LIN {X 88.798,Y 87.967,Z 72.038,A 180.000,B 0.000,C 180.000} C_DIS
LIN {X 88.452,Y 88.283,Z 72.022,A 180.000,B 0.000,C 180.000} C_DIS
LIN {X 88.396,Y 88.335,Z 72.019,A 180.000,B 0.000,C 180.000} C_DIS
LIN {X 88.341,Y 88.389,Z 72.016,A 180.000,B 0.000,C 180.000} C_DIS
LIN {X 88.287,Y 88.444,Z 72.014,A 180.000,B 0.000,C 180.000} C_DIS
LIN {X 87.963,Y 88.776,Z 71.998,A 180.000,B 0.000,C 180.000} C_DIS
LIN {X 87.909,Y 88.831,Z 71.995,A 180.000,B 0.000,C 180.000} C_DIS
LIN {X 87.856,Y 88.887,Z 71.992,A 180.000,B 0.000,C 180.000} C_DIS
LIN {X 87.804,Y 88.944,Z 71.990,A 180.000,B 0.000,C 180.000} C_DIS
LIN {X 87.702,Y 89.060,Z 71.984,A 180.000,B 0.000,C 180.000} C_DIS
LIN {X 87.445,Y 89.355,Z 71.970,A 180.000,B 0.000,C 180.000} C_DIS
LIN {X 87.396,Y 89.412,Z 71.968,A 180.000,B 0.000,C 180.000} C_DIS
LIN {X 87.349,Y 89.471,Z 71.965,A 180.000,B 0.000,C 180.000} C_DIS
LIN {X 87.254,Y 89.593,Z 71.960,A 180.000,B 0.000,C 180.000} C_DIS
LIN {X 87.013,Y 89.903,Z 71.946,A 180.000,B 0.000,C 180.000} C_DIS
LIN {X 86.965,Y 89.965,Z 71.943,A 180.000,B 0.000,C 180.000} C_DIS
LIN {X 86.918,Y 90.027,Z 71.941,A 180.000,B 0.000,C 180.000} C_DIS
LIN {X 86.874,Y 90.090,Z 71.938,A 180.000,B 0.000,C 180.000} C_DIS
LIN {X 86.564,Y 90.537,Z 71.919,A 180.000,B 0.000,C 180.000} C_DIS
LIN {X 86.522,Y 90.601,Z 71.916,A 180.000,B 0.000,C 180.000} C_DIS
LIN {X 86.481,Y 90.665,Z 71.914,A 180.000,B 0.000,C 180.000} C_DIS
LIN {X 86.197,Y 91.129,Z 71.895,A 180.000,B 0.000,C 180.000} C_DIS
LIN {X 86.158,Y 91.194,Z 71.892,A 180.000,B 0.000,C 180.000} C_DIS
LIN {X 86.121,Y 91.260,Z 71.889,A 180.000,B 0.000,C 180.000} C_DIS
LIN {X 86.084,Y 91.327,Z 71.887,A 180.000,B 0.000,C 180.000} C_DIS
LIN {X 85.972,Y 91.535,Z 71.878,A 180.000,B 0.000,C 180.000} C_DIS
LIN {X 85.898,Y 91.673,Z 71.873,A 180.000,B 0.000,C 180.000} C_DIS
LIN {X 85.824,Y 91.810,Z 71.868,A 180.000,B 0.000,C 180.000} C_DIS
LIN {X 85.789,Y 91.879,Z 71.865,A 180.000,B 0.000,C 180.000} C_DIS
LIN {X 85.755,Y 91.949,Z 71.862,A 180.000,B 0.000,C 180.000} C_DIS
LIN {X 85.557,Y 92.373,Z 71.846,A 180.000,B 0.000,C 180.000} C_DIS
LIN {X 85.524,Y 92.444,Z 71.843,A 180.000,B 0.000,C 180.000} C_DIS
LIN {X 85.493,Y 92.514,Z 71.840,A 180.000,B 0.000,C 180.000} C_DIS
LIN {X 85.463,Y 92.585,Z 71.838,A 180.000,B 0.000,C 180.000} C_DIS
LIN {X 85.435,Y 92.656,Z 71.835,A 180.000,B 0.000,C 180.000} C_DIS
LIN {X 85.406,Y 92.727,Z 71.832,A 180.000,B 0.000,C 180.000} C_DIS
LIN {X 85.348,Y 92.873,Z 71.827,A 180.000,B 0.000,C 180.000} C_DIS
LIN {X 85.260,Y 93.091,Z 71.819,A 180.000,B 0.000,C 180.000} C_DIS
LIN {X 85.232,Y 93.163,Z 71.816,A 180.000,B 0.000,C 180.000} C_DIS
LIN {X 85.205,Y 93.235,Z 71.813,A 180.000,B 0.000,C 180.000} C_DIS
LIN {X 85.180,Y 93.308,Z 71.811,A 180.000,B 0.000,C 180.000} C_DIS
LIN {X 85.130,Y 93.456,Z 71.805,A 180.000,B 0.000,C 180.000} C_DIS
LIN {X 85.030,Y 93.751,Z 71.794,A 180.000,B 0.000,C 180.000} C_DIS
LIN {X 85.006,Y 93.825,Z 71.792,A 180.000,B 0.000,C 180.000} C_DIS
LIN {X 84.982,Y 93.898,Z 71.789,A 180.000,B 0.000,C 180.000} C_DIS
LIN {X 84.961,Y 93.974,Z 71.786,A 180.000,B 0.000,C 180.000} C_DIS
LIN {X 84.920,Y 94.125,Z 71.781,A 180.000,B 0.000,C 180.000} C_DIS
LIN {X 84.899,Y 94.200,Z 71.778,A 180.000,B 0.000,C 180.000} C_DIS
LIN {X 84.857,Y 94.352,Z 71.772,A 180.000,B 0.000,C 180.000} C_DIS
LIN {X 84.836,Y 94.428,Z 71.770,A 180.000,B 0.000,C 180.000} C_DIS
LIN {X 84.815,Y 94.504,Z 71.767,A 180.000,B 0.000,C 180.000} C_DIS
LIN {X 84.795,Y 94.578,Z 71.764,A 180.000,B 0.000,C 180.000} C_DIS
LIN {X 84.777,Y 94.653,Z 71.761,A 180.000,B 0.000,C 180.000} C_DIS
LIN {X 84.760,Y 94.728,Z 71.759,A 180.000,B 0.000,C 180.000} C_DIS
LIN {X 84.744,Y 94.804,Z 71.756,A 180.000,B 0.000,C 180.000} C_DIS
LIN {X 84.711,Y 94.958,Z 71.751,A 180.000,B 0.000,C 180.000} C_DIS
LIN {X 84.661,Y 95.187,Z 71.742,A 180.000,B 0.000,C 180.000} C_DIS
LIN {X 84.645,Y 95.263,Z 71.740,A 180.000,B 0.000,C 180.000} C_DIS
LIN {X 84.631,Y 95.339,Z 71.737,A 180.000,B 0.000,C 180.000} C_DIS
LIN {X 84.618,Y 95.415,Z 71.734,A 180.000,B 0.000,C 180.000} C_DIS
LIN {X 84.594,Y 95.571,Z 71.729,A 180.000,B 0.000,C 180.000} C_DIS
LIN {X 84.557,Y 95.803,Z 71.721,A 180.000,B 0.000,C 180.000} C_DIS
LIN {X 84.545,Y 95.880,Z 71.718,A 180.000,B 0.000,C 180.000} C_DIS
LIN {X 84.533,Y 95.956,Z 71.715,A 180.000,B 0.000,C 180.000} C_DIS
LIN {X 84.522,Y 96.033,Z 71.712,A 180.000,B 0.000,C 180.000} C_DIS
LIN {X 84.512,Y 96.111,Z 71.710,A 180.000,B 0.000,C 180.000} C_DIS
LIN {X 84.504,Y 96.189,Z 71.707,A 180.000,B 0.000,C 180.000} C_DIS
LIN {X 84.481,Y 96.424,Z 71.699,A 180.000,B 0.000,C 180.000} C_DIS
LIN {X 84.465,Y 96.580,Z 71.693,A 180.000,B 0.000,C 180.000} C_DIS
LIN {X 84.457,Y 96.659,Z 71.691,A 180.000,B 0.000,C 180.000} C_DIS
LIN {X 84.450,Y 96.736,Z 71.688,A 180.000,B 0.000,C 180.000} C_DIS
LIN {X 84.444,Y 96.813,Z 71.685,A 180.000,B 0.000,C 180.000} C_DIS
LIN {X 84.441,Y 96.891,Z 71.683,A 180.000,B 0.000,C 180.000} C_DIS
LIN {X 84.431,Y 97.125,Z 71.675,A 180.000,B 0.000,C 180.000} C_DIS
LIN {X 84.427,Y 97.204,Z 71.672,A 180.000,B 0.000,C 180.000} C_DIS
LIN {X 84.424,Y 97.283,Z 71.669,A 180.000,B 0.000,C 180.000} C_DIS
LIN {X 84.420,Y 97.361,Z 71.667,A 180.000,B 0.000,C 180.000} C_DIS
LIN {X 84.417,Y 97.439,Z 71.664,A 180.000,B 0.000,C 180.000} C_DIS
LIN {X 84.416,Y 97.517,Z 71.662,A 180.000,B 0.000,C 180.000} C_DIS
LIN {X 84.416,Y 97.595,Z 71.659,A 180.000,B 0.000,C 180.000} C_DIS
LIN {X 84.417,Y 97.674,Z 71.656,A 180.000,B 0.000,C 180.000} C_DIS
LIN {X 84.418,Y 97.752,Z 71.654,A 180.000,B 0.000,C 180.000} C_DIS
LIN {X 84.419,Y 97.830,Z 71.651,A 180.000,B 0.000,C 180.000} C_DIS
LIN {X 84.420,Y 97.909,Z 71.649,A 180.000,B 0.000,C 180.000} C_DIS
LIN {X 84.422,Y 98.065,Z 71.644,A 180.000,B 0.000,C 180.000} C_DIS
LIN {X 84.424,Y 98.222,Z 71.639,A 180.000,B 0.000,C 180.000} C_DIS
LIN {X 84.434,Y 98.378,Z 71.634,A 180.000,B 0.000,C 180.000} C_DIS
LIN {X 84.445,Y 98.534,Z 71.630,A 180.000,B 0.000,C 180.000} C_DIS
LIN {X 84.456,Y 98.691,Z 71.625,A 180.000,B 0.000,C 180.000} C_DIS
LIN {X 84.467,Y 98.849,Z 71.620,A 180.000,B 0.000,C 180.000} C_DIS
LIN {X 84.481,Y 99.004,Z 71.616,A 180.000,B 0.000,C 180.000} C_DIS
LIN {X 84.500,Y 99.159,Z 71.611,A 180.000,B 0.000,C 180.000} C_DIS
LIN {X 84.520,Y 99.315,Z 71.607,A 180.000,B 0.000,C 180.000} C_DIS
LIN {X 84.540,Y 99.471,Z 71.602,A 180.000,B 0.000,C 180.000} C_DIS
LIN {X 84.560,Y 99.626,Z 71.598,A 180.000,B 0.000,C 180.000} C_DIS
LIN {X 84.584,Y 99.781,Z 71.594,A 180.000,B 0.000,C 180.000} C_DIS
LIN {X 84.613,Y 99.935,Z 71.590,A 180.000,B 0.000,C 180.000} C_DIS
LIN {X 84.642,Y 100.090,Z 71.586,A 180.000,B 0.000,C 180.000} C_DIS
LIN {X 84.671,Y 100.245,Z 71.582,A 180.000,B 0.000,C 180.000} C_DIS
LIN {X 84.700,Y 100.399,Z 71.578,A 180.000,B 0.000,C 180.000} C_DIS
LIN {X 84.737,Y 100.552,Z 71.574,A 180.000,B 0.000,C 180.000} C_DIS
LIN {X 84.774,Y 100.704,Z 71.570,A 180.000,B 0.000,C 180.000} C_DIS
LIN {X 84.812,Y 100.857,Z 71.567,A 180.000,B 0.000,C 180.000} C_DIS
LIN {X 84.850,Y 101.009,Z 71.563,A 180.000,B 0.000,C 180.000} C_DIS
LIN {X 84.888,Y 101.161,Z 71.560,A 180.000,B 0.000,C 180.000} C_DIS
LIN {X 84.934,Y 101.312,Z 71.556,A 180.000,B 0.000,C 180.000} C_DIS
LIN {X 84.980,Y 101.462,Z 71.553,A 180.000,B 0.000,C 180.000} C_DIS
LIN {X 85.027,Y 101.613,Z 71.550,A 180.000,B 0.000,C 180.000} C_DIS
LIN {X 85.073,Y 101.763,Z 71.547,A 180.000,B 0.000,C 180.000} C_DIS
LIN {X 85.124,Y 101.911,Z 71.544,A 180.000,B 0.000,C 180.000} C_DIS
LIN {X 85.179,Y 102.059,Z 71.541,A 180.000,B 0.000,C 180.000} C_DIS
LIN {X 85.234,Y 102.206,Z 71.538,A 180.000,B 0.000,C 180.000} C_DIS
LIN {X 85.289,Y 102.354,Z 71.535,A 180.000,B 0.000,C 180.000} C_DIS
LIN {X 85.344,Y 102.501,Z 71.532,A 180.000,B 0.000,C 180.000} C_DIS
LIN {X 85.405,Y 102.646,Z 71.530,A 180.000,B 0.000,C 180.000} C_DIS
LIN {X 85.468,Y 102.790,Z 71.527,A 180.000,B 0.000,C 180.000} C_DIS
LIN {X 85.594,Y 103.079,Z 71.523,A 180.000,B 0.000,C 180.000} C_DIS
LIN {X 85.730,Y 103.362,Z 71.519,A 180.000,B 0.000,C 180.000} C_DIS
LIN {X 85.873,Y 103.643,Z 71.515,A 180.000,B 0.000,C 180.000} C_DIS
LIN {X 86.020,Y 103.921,Z 71.511,A 180.000,B 0.000,C 180.000} C_DIS
LIN {X 86.178,Y 104.193,Z 71.508,A 180.000,B 0.000,C 180.000} C_DIS
LIN {X 86.337,Y 104.465,Z 71.506,A 180.000,B 0.000,C 180.000} C_DIS
LIN {X 86.509,Y 104.729,Z 71.504,A 180.000,B 0.000,C 180.000} C_DIS
LIN {X 86.684,Y 104.991,Z 71.502,A 180.000,B 0.000,C 180.000} C_DIS
LIN {X 86.866,Y 105.248,Z 71.501,A 180.000,B 0.000,C 180.000} C_DIS
LIN {X 87.055,Y 105.500,Z 71.500,A 180.000,B 0.000,C 180.000} C_DIS
LIN {X 87.227,Y 105.724,Z 71.500,A 180.000,B 0.000,C 180.000} C_DIS
; Cutting Move Starts
LIN {X 87.243,Y 105.745,Z 71.500,A 180.000,B 0.000,C 180.000} C_DIS
LIN {X 87.319,Y 105.835,Z 71.500,A 180.000,B 0.000,C 180.000} C_DIS
LIN {X 87.621,Y 106.193,Z 71.500,A 180.000,B 0.000,C 180.000} C_DIS
LIN {X 87.779,Y 106.367,Z 71.500,A 180.000,B 0.000,C 180.000} C_DIS
LIN {X 88.137,Y 106.746,Z 71.500,A 180.000,B 0.000,C 180.000} C_DIS
LIN {X 88.300,Y 106.908,Z 71.500,A 180.000,B 0.000,C 180.000} C_DIS
LIN {X 88.673,Y 107.260,Z 71.500,A 180.000,B 0.000,C 180.000} C_DIS
LIN {X 88.678,Y 107.265,Z 71.500,A 180.000,B 0.000,C 180.000} C_DIS
LIN {X 88.852,Y 107.416,Z 71.500,A 180.000,B 0.000,C 180.000} C_DIS
LIN {X 89.209,Y 107.718,Z 71.500,A 180.000,B 0.000,C 180.000} C_DIS
LIN {X 89.311,Y 107.802,Z 71.500,A 180.000,B 0.000,C 180.000} C_DIS
LIN {X 89.388,Y 107.861,Z 71.500,A 180.000,B 0.000,C 180.000} C_DIS
LIN {X 89.784,Y 108.159,Z 71.500,A 180.000,B 0.000,C 180.000} C_DIS
LIN {X 89.925,Y 108.261,Z 71.500,A 180.000,B 0.000,C 180.000} C_DIS
LIN {X 90.040,Y 108.338,Z 71.500,A 180.000,B 0.000,C 180.000} C_DIS
LIN {X 90.307,Y 108.517,Z 71.500,A 180.000,B 0.000,C 180.000} C_DIS
LIN {X 90.461,Y 108.618,Z 71.500,A 180.000,B 0.000,C 180.000} C_DIS
LIN {X 90.585,Y 108.695,Z 71.500,A 180.000,B 0.000,C 180.000} C_DIS
LIN {X 90.997,Y 108.939,Z 71.500,A 180.000,B 0.000,C 180.000} C_DIS
LIN {X 91.176,Y 109.041,Z 71.500,A 180.000,B 0.000,C 180.000} C_DIS
LIN {X 91.199,Y 109.053,Z 71.500,A 180.000,B 0.000,C 180.000} C_DIS
LIN {X 91.545,Y 109.232,Z 71.500,A 180.000,B 0.000,C 180.000} C_DIS
LIN {X 91.712,Y 109.318,Z 71.500,A 180.000,B 0.000,C 180.000} C_DIS
LIN {X 91.891,Y 109.403,Z 71.500,A 180.000,B 0.000,C 180.000} C_DIS
LIN {X 92.307,Y 109.589,Z 71.500,A 180.000,B 0.000,C 180.000} C_DIS
LIN {X 92.427,Y 109.643,Z 71.500,A 180.000,B 0.000,C 180.000} C_DIS
LIN {X 92.606,Y 109.714,Z 71.500,A 180.000,B 0.000,C 180.000} C_DIS
LIN {X 92.964,Y 109.851,Z 71.500,A 180.000,B 0.000,C 180.000} C_DIS
LIN {X 93.142,Y 109.918,Z 71.500,A 180.000,B 0.000,C 180.000} C_DIS
LIN {X 93.230,Y 109.947,Z 71.500,A 180.000,B 0.000,C 180.000} C_DIS
LIN {X 93.321,Y 109.976,Z 71.500,A 180.000,B 0.000,C 180.000} C_DIS
LIN {X 93.791,Y 110.126,Z 71.500,A 180.000,B 0.000,C 180.000} C_DIS
LIN {X 93.857,Y 110.146,Z 71.500,A 180.000,B 0.000,C 180.000} C_DIS
LIN {X 94.036,Y 110.194,Z 71.500,A 180.000,B 0.000,C 180.000} C_DIS
LIN {X 94.466,Y 110.304,Z 71.500,A 180.000,B 0.000,C 180.000} C_DIS
LIN {X 94.573,Y 110.330,Z 71.500,A 180.000,B 0.000,C 180.000} C_DIS
LIN {X 94.751,Y 110.367,Z 71.500,A 180.000,B 0.000,C 180.000} C_DIS
LIN {X 95.109,Y 110.438,Z 71.500,A 180.000,B 0.000,C 180.000} C_DIS
LIN {X 95.288,Y 110.473,Z 71.500,A 180.000,B 0.000,C 180.000} C_DIS
LIN {X 95.350,Y 110.483,Z 71.500,A 180.000,B 0.000,C 180.000} C_DIS
LIN {X 95.466,Y 110.500,Z 71.500,A 180.000,B 0.000,C 180.000} C_DIS
LIN {X 95.824,Y 110.550,Z 71.500,A 180.000,B 0.000,C 180.000} C_DIS
LIN {X 96.003,Y 110.575,Z 71.500,A 180.000,B 0.000,C 180.000} C_DIS
LIN {X 96.181,Y 110.591,Z 71.500,A 180.000,B 0.000,C 180.000} C_DIS
LIN {X 96.539,Y 110.622,Z 71.500,A 180.000,B 0.000,C 180.000} C_DIS
LIN {X 96.718,Y 110.636,Z 71.500,A 180.000,B 0.000,C 180.000} C_DIS
LIN {X 96.897,Y 110.644,Z 71.500,A 180.000,B 0.000,C 180.000} C_DIS
LIN {X 97.433,Y 110.659,Z 71.500,A 180.000,B 0.000,C 180.000} C_DIS
LIN {X 97.612,Y 110.658,Z 71.500,A 180.000,B 0.000,C 180.000} C_DIS
LIN {X 98.148,Y 110.643,Z 71.500,A 180.000,B 0.000,C 180.000} C_DIS
LIN {X 98.327,Y 110.633,Z 71.500,A 180.000,B 0.000,C 180.000} C_DIS
LIN {X 98.505,Y 110.618,Z 71.500,A 180.000,B 0.000,C 180.000} C_DIS
LIN {X 98.863,Y 110.588,Z 71.500,A 180.000,B 0.000,C 180.000} C_DIS
LIN {X 99.042,Y 110.569,Z 71.500,A 180.000,B 0.000,C 180.000} C_DIS
LIN {X 99.221,Y 110.544,Z 71.500,A 180.000,B 0.000,C 180.000} C_DIS
LIN {X 99.578,Y 110.493,Z 71.500,A 180.000,B 0.000,C 180.000} C_DIS
LIN {X 99.650,Y 110.483,Z 71.500,A 180.000,B 0.000,C 180.000} C_DIS
LIN {X 99.757,Y 110.464,Z 71.500,A 180.000,B 0.000,C 180.000} C_DIS
LIN {X 99.936,Y 110.429,Z 71.500,A 180.000,B 0.000,C 180.000} C_DIS
LIN {X 100.293,Y 110.358,Z 71.500,A 180.000,B 0.000,C 180.000} C_DIS
LIN {X 100.472,Y 110.320,Z 71.500,A 180.000,B 0.000,C 180.000} C_DIS
LIN {X 100.534,Y 110.304,Z 71.500,A 180.000,B 0.000,C 180.000} C_DIS
LIN {X 101.008,Y 110.182,Z 71.500,A 180.000,B 0.000,C 180.000} C_DIS
LIN {X 101.187,Y 110.132,Z 71.500,A 180.000,B 0.000,C 180.000} C_DIS
LIN {X 101.209,Y 110.126,Z 71.500,A 180.000,B 0.000,C 180.000} C_DIS
LIN {X 101.723,Y 109.962,Z 71.500,A 180.000,B 0.000,C 180.000} C_DIS
LIN {X 101.770,Y 109.947,Z 71.500,A 180.000,B 0.000,C 180.000} C_DIS
LIN {X 101.902,Y 109.902,Z 71.500,A 180.000,B 0.000,C 180.000} C_DIS
LIN {X 102.081,Y 109.834,Z 71.500,A 180.000,B 0.000,C 180.000} C_DIS
LIN {X 102.438,Y 109.697,Z 71.500,A 180.000,B 0.000,C 180.000} C_DIS
LIN {X 102.617,Y 109.623,Z 71.500,A 180.000,B 0.000,C 180.000} C_DIS
LIN {X 103.093,Y 109.410,Z 71.500,A 180.000,B 0.000,C 180.000} C_DIS
LIN {X 103.153,Y 109.383,Z 71.500,A 180.000,B 0.000,C 180.000} C_DIS
LIN {X 103.332,Y 109.295,Z 71.500,A 180.000,B 0.000,C 180.000} C_DIS
LIN {X 103.801,Y 109.053,Z 71.500,A 180.000,B 0.000,C 180.000} C_DIS
LIN {X 103.869,Y 109.017,Z 71.500,A 180.000,B 0.000,C 180.000} C_DIS
LIN {X 104.047,Y 108.912,Z 71.500,A 180.000,B 0.000,C 180.000} C_DIS
LIN {X 104.415,Y 108.695,Z 71.500,A 180.000,B 0.000,C 180.000} C_DIS
LIN {X 104.584,Y 108.589,Z 71.500,A 180.000,B 0.000,C 180.000} C_DIS
LIN {X 104.960,Y 108.338,Z 71.500,A 180.000,B 0.000,C 180.000} C_DIS
LIN {X 105.120,Y 108.230,Z 71.500,A 180.000,B 0.000,C 180.000} C_DIS
LIN {X 105.216,Y 108.159,Z 71.500,A 180.000,B 0.000,C 180.000} C_DIS
LIN {X 105.477,Y 107.962,Z 71.500,A 180.000,B 0.000,C 180.000} C_DIS
LIN {X 105.656,Y 107.827,Z 71.500,A 180.000,B 0.000,C 180.000} C_DIS
LIN {X 105.689,Y 107.802,Z 71.500,A 180.000,B 0.000,C 180.000} C_DIS
LIN {X 105.835,Y 107.680,Z 71.500,A 180.000,B 0.000,C 180.000} C_DIS
LIN {X 106.193,Y 107.378,Z 71.500,A 180.000,B 0.000,C 180.000} C_DIS
LIN {X 106.322,Y 107.265,Z 71.500,A 180.000,B 0.000,C 180.000} C_DIS
LIN {X 106.371,Y 107.218,Z 71.500,A 180.000,B 0.000,C 180.000} C_DIS
LIN {X 106.729,Y 106.880,Z 71.500,A 180.000,B 0.000,C 180.000} C_DIS
LIN {X 106.879,Y 106.729,Z 71.500,A 180.000,B 0.000,C 180.000} C_DIS
LIN {X 107.217,Y 106.371,Z 71.500,A 180.000,B 0.000,C 180.000} C_DIS
LIN {X 107.265,Y 106.320,Z 71.500,A 180.000,B 0.000,C 180.000} C_DIS
LIN {X 107.379,Y 106.193,Z 71.500,A 180.000,B 0.000,C 180.000} C_DIS
LIN {X 107.681,Y 105.835,Z 71.500,A 180.000,B 0.000,C 180.000} C_DIS
LIN {X 107.802,Y 105.690,Z 71.500,A 180.000,B 0.000,C 180.000} C_DIS
LIN {X 107.827,Y 105.656,Z 71.500,A 180.000,B 0.000,C 180.000} C_DIS
LIN {X 108.159,Y 105.215,Z 71.500,A 180.000,B 0.000,C 180.000} C_DIS
LIN {X 108.229,Y 105.120,Z 71.500,A 180.000,B 0.000,C 180.000} C_DIS
LIN {X 108.338,Y 104.961,Z 71.500,A 180.000,B 0.000,C 180.000} C_DIS
LIN {X 108.590,Y 104.584,Z 71.500,A 180.000,B 0.000,C 180.000} C_DIS
LIN {X 108.695,Y 104.415,Z 71.500,A 180.000,B 0.000,C 180.000} C_DIS
LIN {X 108.912,Y 104.047,Z 71.500,A 180.000,B 0.000,C 180.000} C_DIS
LIN {X 109.016,Y 103.869,Z 71.500,A 180.000,B 0.000,C 180.000} C_DIS
LIN {X 109.053,Y 103.800,Z 71.500,A 180.000,B 0.000,C 180.000} C_DIS
LIN {X 109.110,Y 103.690,Z 71.500,A 180.000,B 0.000,C 180.000} C_DIS
LIN {X 109.295,Y 103.332,Z 71.500,A 180.000,B 0.000,C 180.000} C_DIS
LIN {X 109.384,Y 103.153,Z 71.500,A 180.000,B 0.000,C 180.000} C_DIS
LIN {X 109.410,Y 103.094,Z 71.500,A 180.000,B 0.000,C 180.000} C_DIS
LIN {X 109.624,Y 102.617,Z 71.500,A 180.000,B 0.000,C 180.000} C_DIS
LIN {X 109.697,Y 102.438,Z 71.500,A 180.000,B 0.000,C 180.000} C_DIS
LIN {X 109.901,Y 101.902,Z 71.500,A 180.000,B 0.000,C 180.000} C_DIS
LIN {X 109.947,Y 101.772,Z 71.500,A 180.000,B 0.000,C 180.000} C_DIS
LIN {X 110.076,Y 101.366,Z 71.500,A 180.000,B 0.000,C 180.000} C_DIS
LIN {X 110.126,Y 101.211,Z 71.500,A 180.000,B 0.000,C 180.000} C_DIS
LIN {X 110.133,Y 101.187,Z 71.500,A 180.000,B 0.000,C 180.000} C_DIS
LIN {X 110.181,Y 101.008,Z 71.500,A 180.000,B 0.000,C 180.000} C_DIS
LIN {X 110.304,Y 100.531,Z 71.500,A 180.000,B 0.000,C 180.000} C_DIS
LIN {X 110.319,Y 100.472,Z 71.500,A 180.000,B 0.000,C 180.000} C_DIS
LIN {X 110.359,Y 100.293,Z 71.500,A 180.000,B 0.000,C 180.000} C_DIS
LIN {X 110.430,Y 99.936,Z 71.500,A 180.000,B 0.000,C 180.000} C_DIS
LIN {X 110.465,Y 99.757,Z 71.500,A 180.000,B 0.000,C 180.000} C_DIS
LIN {X 110.483,Y 99.648,Z 71.500,A 180.000,B 0.000,C 180.000} C_DIS
LIN {X 110.543,Y 99.221,Z 71.500,A 180.000,B 0.000,C 180.000} C_DIS
LIN {X 110.568,Y 99.042,Z 71.500,A 180.000,B 0.000,C 180.000} C_DIS
LIN {X 110.588,Y 98.863,Z 71.500,A 180.000,B 0.000,C 180.000} C_DIS
LIN {X 110.633,Y 98.327,Z 71.500,A 180.000,B 0.000,C 180.000} C_DIS
LIN {X 110.643,Y 98.148,Z 71.500,A 180.000,B 0.000,C 180.000} C_DIS
LIN {X 110.658,Y 97.612,Z 71.500,A 180.000,B 0.000,C 180.000} C_DIS
LIN {X 110.659,Y 97.433,Z 71.500,A 180.000,B 0.000,C 180.000} C_DIS
LIN {X 110.654,Y 97.254,Z 71.500,A 180.000,B 0.000,C 180.000} C_DIS
LIN {X 110.644,Y 96.897,Z 71.500,A 180.000,B 0.000,C 180.000} C_DIS
LIN {X 110.637,Y 96.718,Z 71.500,A 180.000,B 0.000,C 180.000} C_DIS
LIN {X 110.622,Y 96.539,Z 71.500,A 180.000,B 0.000,C 180.000} C_DIS
LIN {X 110.592,Y 96.181,Z 71.500,A 180.000,B 0.000,C 180.000} C_DIS
LIN {X 110.574,Y 96.003,Z 71.500,A 180.000,B 0.000,C 180.000} C_DIS
LIN {X 110.550,Y 95.824,Z 71.500,A 180.000,B 0.000,C 180.000} C_DIS
LIN {X 110.483,Y 95.352,Z 71.500,A 180.000,B 0.000,C 180.000} C_DIS
LIN {X 110.473,Y 95.288,Z 71.500,A 180.000,B 0.000,C 180.000} C_DIS
LIN {X 110.438,Y 95.109,Z 71.500,A 180.000,B 0.000,C 180.000} C_DIS
LIN {X 110.367,Y 94.751,Z 71.500,A 180.000,B 0.000,C 180.000} C_DIS
LIN {X 110.330,Y 94.573,Z 71.500,A 180.000,B 0.000,C 180.000} C_DIS
LIN {X 110.304,Y 94.469,Z 71.500,A 180.000,B 0.000,C 180.000} C_DIS
LIN {X 110.193,Y 94.036,Z 71.500,A 180.000,B 0.000,C 180.000} C_DIS
LIN {X 110.146,Y 93.857,Z 71.500,A 180.000,B 0.000,C 180.000} C_DIS
LIN {X 110.126,Y 93.789,Z 71.500,A 180.000,B 0.000,C 180.000} C_DIS
LIN {X 110.090,Y 93.679,Z 71.500,A 180.000,B 0.000,C 180.000} C_DIS
LIN {X 109.947,Y 93.228,Z 71.500,A 180.000,B 0.000,C 180.000} C_DIS
LIN {X 109.918,Y 93.142,Z 71.500,A 180.000,B 0.000,C 180.000} C_DIS
LIN {X 109.850,Y 92.964,Z 71.500,A 180.000,B 0.000,C 180.000} C_DIS
LIN {X 109.714,Y 92.606,Z 71.500,A 180.000,B 0.000,C 180.000} C_DIS
LIN {X 109.643,Y 92.427,Z 71.500,A 180.000,B 0.000,C 180.000} C_DIS
LIN {X 109.589,Y 92.306,Z 71.500,A 180.000,B 0.000,C 180.000} C_DIS
LIN {X 109.403,Y 91.891,Z 71.500,A 180.000,B 0.000,C 180.000} C_DIS
LIN {X 109.318,Y 91.712,Z 71.500,A 180.000,B 0.000,C 180.000} C_DIS
LIN {X 109.133,Y 91.355,Z 71.500,A 180.000,B 0.000,C 180.000} C_DIS
LIN {X 109.053,Y 91.200,Z 71.500,A 180.000,B 0.000,C 180.000} C_DIS
LIN {X 109.040,Y 91.176,Z 71.500,A 180.000,B 0.000,C 180.000} C_DIS
LIN {X 108.939,Y 90.997,Z 71.500,A 180.000,B 0.000,C 180.000} C_DIS
LIN {X 108.695,Y 90.585,Z 71.500,A 180.000,B 0.000,C 180.000} C_DIS
LIN {X 108.619,Y 90.461,Z 71.500,A 180.000,B 0.000,C 180.000} C_DIS
LIN {X 108.517,Y 90.307,Z 71.500,A 180.000,B 0.000,C 180.000} C_DIS
LIN {X 108.338,Y 90.039,Z 71.500,A 180.000,B 0.000,C 180.000} C_DIS
LIN {X 108.261,Y 89.925,Z 71.500,A 180.000,B 0.000,C 180.000} C_DIS
LIN {X 108.159,Y 89.785,Z 71.500,A 180.000,B 0.000,C 180.000} C_DIS
LIN {X 107.860,Y 89.388,Z 71.500,A 180.000,B 0.000,C 180.000} C_DIS
LIN {X 107.802,Y 89.310,Z 71.500,A 180.000,B 0.000,C 180.000} C_DIS
LIN {X 107.719,Y 89.209,Z 71.500,A 180.000,B 0.000,C 180.000} C_DIS
LIN {X 107.417,Y 88.852,Z 71.500,A 180.000,B 0.000,C 180.000} C_DIS
LIN {X 107.265,Y 88.680,Z 71.500,A 180.000,B 0.000,C 180.000} C_DIS
LIN {X 107.259,Y 88.673,Z 71.500,A 180.000,B 0.000,C 180.000} C_DIS
LIN {X 107.086,Y 88.491,Z 71.500,A 180.000,B 0.000,C 180.000} C_DIS
LIN {X 106.908,Y 88.301,Z 71.500,A 180.000,B 0.000,C 180.000} C_DIS
LIN {X 106.747,Y 88.137,Z 71.500,A 180.000,B 0.000,C 180.000} C_DIS
LIN {X 106.369,Y 87.779,Z 71.500,A 180.000,B 0.000,C 180.000} C_DIS
LIN {X 106.193,Y 87.622,Z 71.500,A 180.000,B 0.000,C 180.000} C_DIS
LIN {X 105.835,Y 87.320,Z 71.500,A 180.000,B 0.000,C 180.000} C_DIS
LIN {X 105.744,Y 87.243,Z 71.500,A 180.000,B 0.000,C 180.000} C_DIS
LIN {X 105.656,Y 87.173,Z 71.500,A 180.000,B 0.000,C 180.000} C_DIS
LIN {X 105.512,Y 87.064,Z 71.500,A 180.000,B 0.000,C 180.000} C_DIS
LIN {X 105.275,Y 86.885,Z 71.500,A 180.000,B 0.000,C 180.000} C_DIS
LIN {X 105.192,Y 86.824,Z 71.500,A 180.000,B 0.000,C 180.000} C_DIS
LIN {X 105.120,Y 86.770,Z 71.500,A 180.000,B 0.000,C 180.000} C_DIS
LIN {X 105.027,Y 86.707,Z 71.500,A 180.000,B 0.000,C 180.000} C_DIS
LIN {X 104.584,Y 86.411,Z 71.500,A 180.000,B 0.000,C 180.000} C_DIS
LIN {X 104.488,Y 86.349,Z 71.500,A 180.000,B 0.000,C 180.000} C_DIS
LIN {X 104.405,Y 86.299,Z 71.500,A 180.000,B 0.000,C 180.000} C_DIS
LIN {X 104.047,Y 86.088,Z 71.500,A 180.000,B 0.000,C 180.000} C_DIS
LIN {X 103.884,Y 85.992,Z 71.500,A 180.000,B 0.000,C 180.000} C_DIS
LIN {X 103.869,Y 85.983,Z 71.500,A 180.000,B 0.000,C 180.000} C_DIS
LIN {X 103.690,Y 85.890,Z 71.500,A 180.000,B 0.000,C 180.000} C_DIS
LIN {X 103.332,Y 85.705,Z 71.500,A 180.000,B 0.000,C 180.000} C_DIS
LIN {X 103.189,Y 85.634,Z 71.500,A 180.000,B 0.000,C 180.000} C_DIS
LIN {X 103.153,Y 85.617,Z 71.500,A 180.000,B 0.000,C 180.000} C_DIS
LIN {X 102.975,Y 85.537,Z 71.500,A 180.000,B 0.000,C 180.000} C_DIS
LIN {X 102.617,Y 85.377,Z 71.500,A 180.000,B 0.000,C 180.000} C_DIS
LIN {X 102.438,Y 85.303,Z 71.500,A 180.000,B 0.000,C 180.000} C_DIS
LIN {X 102.081,Y 85.166,Z 71.500,A 180.000,B 0.000,C 180.000} C_DIS
LIN {X 101.902,Y 85.098,Z 71.500,A 180.000,B 0.000,C 180.000} C_DIS
LIN {X 101.901,Y 85.098,Z 71.500,A 180.000,B 0.000,C 180.000} C_DIS
LIN {X 101.723,Y 85.038,Z 71.500,A 180.000,B 0.000,C 180.000} C_DIS
LIN {X 101.349,Y 84.919,Z 71.500,A 180.000,B 0.000,C 180.000} C_DIS
LIN {X 101.187,Y 84.868,Z 71.500,A 180.000,B 0.000,C 180.000} C_DIS
LIN {X 101.008,Y 84.818,Z 71.500,A 180.000,B 0.000,C 180.000} C_DIS
LIN {X 100.651,Y 84.726,Z 71.500,A 180.000,B 0.000,C 180.000} C_DIS
LIN {X 100.472,Y 84.680,Z 71.500,A 180.000,B 0.000,C 180.000} C_DIS
LIN {X 100.293,Y 84.642,Z 71.500,A 180.000,B 0.000,C 180.000} C_DIS
LIN {X 99.887,Y 84.561,Z 71.500,A 180.000,B 0.000,C 180.000} C_DIS
LIN {X 99.757,Y 84.536,Z 71.500,A 180.000,B 0.000,C 180.000} C_DIS
LIN {X 99.578,Y 84.507,Z 71.500,A 180.000,B 0.000,C 180.000} C_DIS
LIN {X 99.221,Y 84.456,Z 71.500,A 180.000,B 0.000,C 180.000} C_DIS
LIN {X 99.042,Y 84.431,Z 71.500,A 180.000,B 0.000,C 180.000} C_DIS
LIN {X 98.863,Y 84.412,Z 71.500,A 180.000,B 0.000,C 180.000} C_DIS
LIN {X 98.505,Y 84.382,Z 71.500,A 180.000,B 0.000,C 180.000} C_DIS
LIN {X 98.327,Y 84.367,Z 71.500,A 180.000,B 0.000,C 180.000} C_DIS
LIN {X 98.148,Y 84.357,Z 71.500,A 180.000,B 0.000,C 180.000} C_DIS
LIN {X 97.612,Y 84.342,Z 71.500,A 180.000,B 0.000,C 180.000} C_DIS
LIN {X 97.433,Y 84.341,Z 71.500,A 180.000,B 0.000,C 180.000} C_DIS
LIN {X 96.897,Y 84.356,Z 71.500,A 180.000,B 0.000,C 180.000} C_DIS
LIN {X 96.718,Y 84.364,Z 71.500,A 180.000,B 0.000,C 180.000} C_DIS
LIN {X 96.539,Y 84.378,Z 71.500,A 180.000,B 0.000,C 180.000} C_DIS
LIN {X 96.181,Y 84.409,Z 71.500,A 180.000,B 0.000,C 180.000} C_DIS
LIN {X 96.003,Y 84.425,Z 71.500,A 180.000,B 0.000,C 180.000} C_DIS
LIN {X 95.824,Y 84.450,Z 71.500,A 180.000,B 0.000,C 180.000} C_DIS
LIN {X 95.466,Y 84.500,Z 71.500,A 180.000,B 0.000,C 180.000} C_DIS
LIN {X 95.288,Y 84.527,Z 71.500,A 180.000,B 0.000,C 180.000} C_DIS
LIN {X 95.113,Y 84.561,Z 71.500,A 180.000,B 0.000,C 180.000} C_DIS
LIN {X 94.751,Y 84.633,Z 71.500,A 180.000,B 0.000,C 180.000} C_DIS
LIN {X 94.573,Y 84.670,Z 71.500,A 180.000,B 0.000,C 180.000} C_DIS
LIN {X 94.394,Y 84.714,Z 71.500,A 180.000,B 0.000,C 180.000} C_DIS
LIN {X 94.036,Y 84.806,Z 71.500,A 180.000,B 0.000,C 180.000} C_DIS
LIN {X 93.857,Y 84.854,Z 71.500,A 180.000,B 0.000,C 180.000} C_DIS
LIN {X 93.679,Y 84.910,Z 71.500,A 180.000,B 0.000,C 180.000} C_DIS
LIN {X 93.321,Y 85.024,Z 71.500,A 180.000,B 0.000,C 180.000} C_DIS
LIN {X 93.142,Y 85.082,Z 71.500,A 180.000,B 0.000,C 180.000} C_DIS
LIN {X 93.099,Y 85.098,Z 71.500,A 180.000,B 0.000,C 180.000} C_DIS
LIN {X 92.964,Y 85.149,Z 71.500,A 180.000,B 0.000,C 180.000} C_DIS
LIN {X 92.606,Y 85.286,Z 71.500,A 180.000,B 0.000,C 180.000} C_DIS
LIN {X 92.427,Y 85.357,Z 71.500,A 180.000,B 0.000,C 180.000} C_DIS
LIN {X 92.249,Y 85.437,Z 71.500,A 180.000,B 0.000,C 180.000} C_DIS
LIN {X 91.891,Y 85.597,Z 71.500,A 180.000,B 0.000,C 180.000} C_DIS
LIN {X 91.811,Y 85.634,Z 71.500,A 180.000,B 0.000,C 180.000} C_DIS
LIN {X 91.712,Y 85.682,Z 71.500,A 180.000,B 0.000,C 180.000} C_DIS
LIN {X 91.459,Y 85.813,Z 71.500,A 180.000,B 0.000,C 180.000} C_DIS
LIN {X 91.355,Y 85.867,Z 71.500,A 180.000,B 0.000,C 180.000} C_DIS
LIN {X 91.176,Y 85.959,Z 71.500,A 180.000,B 0.000,C 180.000} C_DIS
LIN {X 91.116,Y 85.992,Z 71.500,A 180.000,B 0.000,C 180.000} C_DIS
LIN {X 90.997,Y 86.061,Z 71.500,A 180.000,B 0.000,C 180.000} C_DIS
LIN {X 90.640,Y 86.272,Z 71.500,A 180.000,B 0.000,C 180.000} C_DIS
LIN {X 90.512,Y 86.349,Z 71.500,A 180.000,B 0.000,C 180.000} C_DIS
LIN {X 90.461,Y 86.382,Z 71.500,A 180.000,B 0.000,C 180.000} C_DIS
LIN {X 90.282,Y 86.500,Z 71.500,A 180.000,B 0.000,C 180.000} C_DIS
LIN {X 89.973,Y 86.707,Z 71.500,A 180.000,B 0.000,C 180.000} C_DIS
LIN {X 89.925,Y 86.739,Z 71.500,A 180.000,B 0.000,C 180.000} C_DIS
LIN {X 89.746,Y 86.870,Z 71.500,A 180.000,B 0.000,C 180.000} C_DIS
LIN {X 89.388,Y 87.139,Z 71.500,A 180.000,B 0.000,C 180.000} C_DIS
LIN {X 89.256,Y 87.243,Z 71.500,A 180.000,B 0.000,C 180.000} C_DIS
LIN {X 89.209,Y 87.282,Z 71.500,A 180.000,B 0.000,C 180.000} C_DIS
LIN {X 88.832,Y 87.601,Z 71.500,A 180.000,B 0.000,C 180.000} C_DIS
LIN {X 88.673,Y 87.740,Z 71.500,A 180.000,B 0.000,C 180.000} C_DIS
LIN {X 88.253,Y 88.137,Z 71.500,A 180.000,B 0.000,C 180.000} C_DIS
LIN {X 88.137,Y 88.254,Z 71.500,A 180.000,B 0.000,C 180.000} C_DIS
LIN {X 87.779,Y 88.633,Z 71.500,A 180.000,B 0.000,C 180.000} C_DIS
LIN {X 87.741,Y 88.673,Z 71.500,A 180.000,B 0.000,C 180.000} C_DIS
LIN {X 87.601,Y 88.831,Z 71.500,A 180.000,B 0.000,C 180.000} C_DIS
LIN {X 87.281,Y 89.209,Z 71.500,A 180.000,B 0.000,C 180.000} C_DIS
LIN {X 87.243,Y 89.255,Z 71.500,A 180.000,B 0.000,C 180.000} C_DIS
LIN {X 87.140,Y 89.388,Z 71.500,A 180.000,B 0.000,C 180.000} C_DIS
LIN {X 86.870,Y 89.746,Z 71.500,A 180.000,B 0.000,C 180.000} C_DIS
LIN {X 86.739,Y 89.925,Z 71.500,A 180.000,B 0.000,C 180.000} C_DIS
LIN {X 86.707,Y 89.973,Z 71.500,A 180.000,B 0.000,C 180.000} C_DIS
LIN {X 86.500,Y 90.282,Z 71.500,A 180.000,B 0.000,C 180.000} C_DIS
LIN {X 86.381,Y 90.461,Z 71.500,A 180.000,B 0.000,C 180.000} C_DIS
LIN {X 86.349,Y 90.511,Z 71.500,A 180.000,B 0.000,C 180.000} C_DIS
LIN {X 86.272,Y 90.640,Z 71.500,A 180.000,B 0.000,C 180.000} C_DIS
LIN {X 86.061,Y 90.997,Z 71.500,A 180.000,B 0.000,C 180.000} C_DIS
LIN {X 85.992,Y 91.118,Z 71.500,A 180.000,B 0.000,C 180.000} C_DIS
LIN {X 85.960,Y 91.176,Z 71.500,A 180.000,B 0.000,C 180.000} C_DIS
LIN {X 85.867,Y 91.355,Z 71.500,A 180.000,B 0.000,C 180.000} C_DIS
LIN {X 85.682,Y 91.712,Z 71.500,A 180.000,B 0.000,C 180.000} C_DIS
LIN {X 85.634,Y 91.809,Z 71.500,A 180.000,B 0.000,C 180.000} C_DIS
LIN {X 85.597,Y 91.891,Z 71.500,A 180.000,B 0.000,C 180.000} C_DIS
LIN {X 85.437,Y 92.249,Z 71.500,A 180.000,B 0.000,C 180.000} C_DIS
LIN {X 85.357,Y 92.427,Z 71.500,A 180.000,B 0.000,C 180.000} C_DIS
LIN {X 85.286,Y 92.606,Z 71.500,A 180.000,B 0.000,C 180.000} C_DIS
LIN {X 85.098,Y 93.100,Z 71.500,A 180.000,B 0.000,C 180.000} C_DIS
LIN {X 85.082,Y 93.142,Z 71.500,A 180.000,B 0.000,C 180.000} C_DIS
LIN {X 85.023,Y 93.321,Z 71.500,A 180.000,B 0.000,C 180.000} C_DIS
LIN {X 84.910,Y 93.679,Z 71.500,A 180.000,B 0.000,C 180.000} C_DIS
LIN {X 84.854,Y 93.857,Z 71.500,A 180.000,B 0.000,C 180.000} C_DIS
LIN {X 84.807,Y 94.036,Z 71.500,A 180.000,B 0.000,C 180.000} C_DIS
LIN {X 84.715,Y 94.394,Z 71.500,A 180.000,B 0.000,C 180.000} C_DIS
LIN {X 84.670,Y 94.573,Z 71.500,A 180.000,B 0.000,C 180.000} C_DIS
LIN {X 84.633,Y 94.751,Z 71.500,A 180.000,B 0.000,C 180.000} C_DIS
LIN {X 84.561,Y 95.109,Z 71.500,A 180.000,B 0.000,C 180.000} C_DIS
LIN {X 84.527,Y 95.288,Z 71.500,A 180.000,B 0.000,C 180.000} C_DIS
LIN {X 84.501,Y 95.466,Z 71.500,A 180.000,B 0.000,C 180.000} C_DIS
LIN {X 84.450,Y 95.824,Z 71.500,A 180.000,B 0.000,C 180.000} C_DIS
LIN {X 84.432,Y 95.959,Z 71.500,A 180.000,B 0.000,C 180.000} C_DIS
LIN {X 84.426,Y 96.003,Z 71.500,A 180.000,B 0.000,C 180.000} C_DIS
LIN {X 84.408,Y 96.181,Z 71.500,A 180.000,B 0.000,C 180.000} C_DIS
LIN {X 84.383,Y 96.485,Z 71.500,A 180.000,B 0.000,C 180.000} C_DIS
LIN {X 84.378,Y 96.539,Z 71.500,A 180.000,B 0.000,C 180.000} C_DIS
LIN {X 84.363,Y 96.718,Z 71.500,A 180.000,B 0.000,C 180.000} C_DIS
LIN {X 84.356,Y 96.897,Z 71.500,A 180.000,B 0.000,C 180.000} C_DIS
LIN {X 84.346,Y 97.254,Z 71.500,A 180.000,B 0.000,C 180.000} C_DIS
LIN {X 84.341,Y 97.433,Z 71.500,A 180.000,B 0.000,C 180.000} C_DIS
LIN {X 84.342,Y 97.612,Z 71.500,A 180.000,B 0.000,C 180.000} C_DIS
LIN {X 84.357,Y 98.148,Z 71.500,A 180.000,B 0.000,C 180.000} C_DIS
LIN {X 84.367,Y 98.327,Z 71.500,A 180.000,B 0.000,C 180.000} C_DIS
LIN {X 84.412,Y 98.863,Z 71.500,A 180.000,B 0.000,C 180.000} C_DIS
LIN {X 84.432,Y 99.042,Z 71.500,A 180.000,B 0.000,C 180.000} C_DIS
LIN {X 84.457,Y 99.221,Z 71.500,A 180.000,B 0.000,C 180.000} C_DIS
LIN {X 84.507,Y 99.578,Z 71.500,A 180.000,B 0.000,C 180.000} C_DIS
LIN {X 84.535,Y 99.757,Z 71.500,A 180.000,B 0.000,C 180.000} C_DIS
LIN {X 84.561,Y 99.891,Z 71.500,A 180.000,B 0.000,C 180.000} C_DIS
LIN {X 84.641,Y 100.293,Z 71.500,A 180.000,B 0.000,C 180.000} C_DIS
LIN {X 84.681,Y 100.472,Z 71.500,A 180.000,B 0.000,C 180.000} C_DIS
LIN {X 84.727,Y 100.651,Z 71.500,A 180.000,B 0.000,C 180.000} C_DIS
LIN {X 84.819,Y 101.008,Z 71.500,A 180.000,B 0.000,C 180.000} C_DIS
LIN {X 84.867,Y 101.187,Z 71.500,A 180.000,B 0.000,C 180.000} C_DIS
LIN {X 84.919,Y 101.351,Z 71.500,A 180.000,B 0.000,C 180.000} C_DIS
LIN {X 85.038,Y 101.723,Z 71.500,A 180.000,B 0.000,C 180.000} C_DIS
LIN {X 85.098,Y 101.900,Z 71.500,A 180.000,B 0.000,C 180.000} C_DIS
LIN {X 85.303,Y 102.438,Z 71.500,A 180.000,B 0.000,C 180.000} C_DIS
LIN {X 85.376,Y 102.617,Z 71.500,A 180.000,B 0.000,C 180.000} C_DIS
LIN {X 85.536,Y 102.975,Z 71.500,A 180.000,B 0.000,C 180.000} C_DIS
LIN {X 85.616,Y 103.153,Z 71.500,A 180.000,B 0.000,C 180.000} C_DIS
LIN {X 85.634,Y 103.191,Z 71.500,A 180.000,B 0.000,C 180.000} C_DIS
LIN {X 85.705,Y 103.332,Z 71.500,A 180.000,B 0.000,C 180.000} C_DIS
LIN {X 85.890,Y 103.690,Z 71.500,A 180.000,B 0.000,C 180.000} C_DIS
LIN {X 85.984,Y 103.869,Z 71.500,A 180.000,B 0.000,C 180.000} C_DIS
LIN {X 85.992,Y 103.882,Z 71.500,A 180.000,B 0.000,C 180.000} C_DIS
LIN {X 86.088,Y 104.047,Z 71.500,A 180.000,B 0.000,C 180.000} C_DIS
LIN {X 86.299,Y 104.405,Z 71.500,A 180.000,B 0.000,C 180.000} C_DIS
LIN {X 86.349,Y 104.489,Z 71.500,A 180.000,B 0.000,C 180.000} C_DIS
LIN {X 86.410,Y 104.584,Z 71.500,A 180.000,B 0.000,C 180.000} C_DIS
LIN {X 86.707,Y 105.027,Z 71.500,A 180.000,B 0.000,C 180.000} C_DIS
LIN {X 86.771,Y 105.120,Z 71.500,A 180.000,B 0.000,C 180.000} C_DIS
LIN {X 86.885,Y 105.274,Z 71.500,A 180.000,B 0.000,C 180.000} C_DIS
LIN {X 87.173,Y 105.656,Z 71.500,A 180.000,B 0.000,C 180.000} C_DIS
LIN {X 87.227,Y 105.724,Z 71.500,A 180.000,B 0.000,C 180.000} C_DIS
; Link Move Starts
LIN {X 87.425,Y 105.961,Z 71.500,A 180.000,B 0.000,C 180.000} C_DIS
LIN {X 87.627,Y 106.201,Z 71.499,A 180.000,B 0.000,C 180.000} C_DIS
LIN {X 87.823,Y 106.415,Z 71.498,A 180.000,B 0.000,C 180.000} C_DIS
LIN {X 88.039,Y 106.644,Z 71.496,A 180.000,B 0.000,C 180.000} C_DIS
LIN {X 88.246,Y 106.860,Z 71.494,A 180.000,B 0.000,C 180.000} C_DIS
LIN {X 88.467,Y 107.070,Z 71.492,A 180.000,B 0.000,C 180.000} C_DIS
LIN {X 88.688,Y 107.282,Z 71.489,A 180.000,B 0.000,C 180.000} C_DIS
LIN {X 88.914,Y 107.477,Z 71.486,A 180.000,B 0.000,C 180.000} C_DIS
LIN {X 89.151,Y 107.680,Z 71.482,A 180.000,B 0.000,C 180.000} C_DIS
LIN {X 89.377,Y 107.866,Z 71.478,A 180.000,B 0.000,C 180.000} C_DIS
LIN {X 89.627,Y 108.056,Z 71.474,A 180.000,B 0.000,C 180.000} C_DIS
LIN {X 89.863,Y 108.236,Z 71.469,A 180.000,B 0.000,C 180.000} C_DIS
LIN {X 89.990,Y 108.323,Z 71.466,A 180.000,B 0.000,C 180.000} C_DIS
LIN {X 90.117,Y 108.410,Z 71.464,A 180.000,B 0.000,C 180.000} C_DIS
LIN {X 90.245,Y 108.497,Z 71.461,A 180.000,B 0.000,C 180.000} C_DIS
LIN {X 90.374,Y 108.584,Z 71.458,A 180.000,B 0.000,C 180.000} C_DIS
LIN {X 90.497,Y 108.666,Z 71.455,A 180.000,B 0.000,C 180.000} C_DIS
LIN {X 90.623,Y 108.744,Z 71.452,A 180.000,B 0.000,C 180.000} C_DIS
LIN {X 90.757,Y 108.825,Z 71.449,A 180.000,B 0.000,C 180.000} C_DIS
LIN {X 90.892,Y 108.906,Z 71.446,A 180.000,B 0.000,C 180.000} C_DIS
LIN {X 91.019,Y 108.983,Z 71.443,A 180.000,B 0.000,C 180.000} C_DIS
LIN {X 91.148,Y 109.058,Z 71.439,A 180.000,B 0.000,C 180.000} C_DIS
LIN {X 91.283,Y 109.130,Z 71.436,A 180.000,B 0.000,C 180.000} C_DIS
LIN {X 91.419,Y 109.202,Z 71.433,A 180.000,B 0.000,C 180.000} C_DIS
LIN {X 91.558,Y 109.276,Z 71.429,A 180.000,B 0.000,C 180.000} C_DIS
LIN {X 91.697,Y 109.350,Z 71.425,A 180.000,B 0.000,C 180.000} C_DIS
LIN {X 91.828,Y 109.415,Z 71.422,A 180.000,B 0.000,C 180.000} C_DIS
LIN {X 91.960,Y 109.476,Z 71.418,A 180.000,B 0.000,C 180.000} C_DIS
LIN {X 92.103,Y 109.542,Z 71.414,A 180.000,B 0.000,C 180.000} C_DIS
LIN {X 92.246,Y 109.608,Z 71.410,A 180.000,B 0.000,C 180.000} C_DIS
LIN {X 92.382,Y 109.671,Z 71.406,A 180.000,B 0.000,C 180.000} C_DIS
LIN {X 92.519,Y 109.730,Z 71.402,A 180.000,B 0.000,C 180.000} C_DIS
LIN {X 92.662,Y 109.787,Z 71.398,A 180.000,B 0.000,C 180.000} C_DIS
LIN {X 92.805,Y 109.843,Z 71.393,A 180.000,B 0.000,C 180.000} C_DIS
LIN {X 92.950,Y 109.901,Z 71.389,A 180.000,B 0.000,C 180.000} C_DIS
LIN {X 93.096,Y 109.959,Z 71.384,A 180.000,B 0.000,C 180.000} C_DIS
LIN {X 93.235,Y 110.007,Z 71.380,A 180.000,B 0.000,C 180.000} C_DIS
LIN {X 93.374,Y 110.053,Z 71.376,A 180.000,B 0.000,C 180.000} C_DIS
LIN {X 93.523,Y 110.103,Z 71.371,A 180.000,B 0.000,C 180.000} C_DIS
LIN {X 93.673,Y 110.153,Z 71.366,A 180.000,B 0.000,C 180.000} C_DIS
LIN {X 93.815,Y 110.201,Z 71.362,A 180.000,B 0.000,C 180.000} C_DIS
LIN {X 93.959,Y 110.243,Z 71.357,A 180.000,B 0.000,C 180.000} C_DIS
LIN {X 94.107,Y 110.283,Z 71.352,A 180.000,B 0.000,C 180.000} C_DIS
LIN {X 94.256,Y 110.324,Z 71.347,A 180.000,B 0.000,C 180.000} C_DIS
LIN {X 94.401,Y 110.364,Z 71.342,A 180.000,B 0.000,C 180.000} C_DIS
LIN {X 94.546,Y 110.402,Z 71.337,A 180.000,B 0.000,C 180.000} C_DIS
LIN {X 94.621,Y 110.419,Z 71.335,A 180.000,B 0.000,C 180.000} C_DIS
LIN {X 94.696,Y 110.436,Z 71.332,A 180.000,B 0.000,C 180.000} C_DIS
LIN {X 94.771,Y 110.452,Z 71.329,A 180.000,B 0.000,C 180.000} C_DIS
LIN {X 94.923,Y 110.484,Z 71.324,A 180.000,B 0.000,C 180.000} C_DIS
LIN {X 95.000,Y 110.501,Z 71.322,A 180.000,B 0.000,C 180.000} C_DIS
LIN {X 95.077,Y 110.518,Z 71.319,A 180.000,B 0.000,C 180.000} C_DIS
LIN {X 95.154,Y 110.534,Z 71.316,A 180.000,B 0.000,C 180.000} C_DIS
LIN {X 95.226,Y 110.549,Z 71.314,A 180.000,B 0.000,C 180.000} C_DIS
LIN {X 95.298,Y 110.564,Z 71.311,A 180.000,B 0.000,C 180.000} C_DIS
LIN {X 95.371,Y 110.576,Z 71.308,A 180.000,B 0.000,C 180.000} C_DIS
LIN {X 95.443,Y 110.588,Z 71.306,A 180.000,B 0.000,C 180.000} C_DIS
LIN {X 95.599,Y 110.612,Z 71.300,A 180.000,B 0.000,C 180.000} C_DIS
LIN {X 95.827,Y 110.648,Z 71.292,A 180.000,B 0.000,C 180.000} C_DIS
LIN {X 95.900,Y 110.660,Z 71.290,A 180.000,B 0.000,C 180.000} C_DIS
LIN {X 95.973,Y 110.671,Z 71.287,A 180.000,B 0.000,C 180.000} C_DIS
LIN {X 96.046,Y 110.681,Z 71.285,A 180.000,B 0.000,C 180.000} C_DIS
LIN {X 96.124,Y 110.689,Z 71.282,A 180.000,B 0.000,C 180.000} C_DIS
LIN {X 96.281,Y 110.704,Z 71.276,A 180.000,B 0.000,C 180.000} C_DIS
LIN {X 96.359,Y 110.712,Z 71.274,A 180.000,B 0.000,C 180.000} C_DIS
LIN {X 96.515,Y 110.728,Z 71.268,A 180.000,B 0.000,C 180.000} C_DIS
LIN {X 96.592,Y 110.736,Z 71.265,A 180.000,B 0.000,C 180.000} C_DIS
LIN {X 96.670,Y 110.744,Z 71.263,A 180.000,B 0.000,C 180.000} C_DIS
LIN {X 96.744,Y 110.750,Z 71.260,A 180.000,B 0.000,C 180.000} C_DIS
LIN {X 96.819,Y 110.755,Z 71.258,A 180.000,B 0.000,C 180.000} C_DIS
LIN {X 96.893,Y 110.759,Z 71.255,A 180.000,B 0.000,C 180.000} C_DIS
LIN {X 96.967,Y 110.762,Z 71.252,A 180.000,B 0.000,C 180.000} C_DIS
LIN {X 97.124,Y 110.769,Z 71.247,A 180.000,B 0.000,C 180.000} C_DIS
LIN {X 97.357,Y 110.779,Z 71.239,A 180.000,B 0.000,C 180.000} C_DIS
LIN {X 97.433,Y 110.783,Z 71.236,A 180.000,B 0.000,C 180.000} C_DIS
LIN {X 97.509,Y 110.785,Z 71.233,A 180.000,B 0.000,C 180.000} C_DIS
LIN {X 97.585,Y 110.785,Z 71.231,A 180.000,B 0.000,C 180.000} C_DIS
LIN {X 97.739,Y 110.783,Z 71.225,A 180.000,B 0.000,C 180.000} C_DIS
LIN {X 98.046,Y 110.779,Z 71.215,A 180.000,B 0.000,C 180.000} C_DIS
LIN {X 98.123,Y 110.778,Z 71.212,A 180.000,B 0.000,C 180.000} C_DIS
LIN {X 98.200,Y 110.777,Z 71.209,A 180.000,B 0.000,C 180.000} C_DIS
LIN {X 98.276,Y 110.774,Z 71.207,A 180.000,B 0.000,C 180.000} C_DIS
LIN {X 98.352,Y 110.769,Z 71.204,A 180.000,B 0.000,C 180.000} C_DIS
LIN {X 98.818,Y 110.738,Z 71.188,A 180.000,B 0.000,C 180.000} C_DIS
LIN {X 98.892,Y 110.733,Z 71.185,A 180.000,B 0.000,C 180.000} C_DIS
LIN {X 98.967,Y 110.727,Z 71.182,A 180.000,B 0.000,C 180.000} C_DIS
LIN {X 99.041,Y 110.720,Z 71.180,A 180.000,B 0.000,C 180.000} C_DIS
LIN {X 99.115,Y 110.711,Z 71.177,A 180.000,B 0.000,C 180.000} C_DIS
LIN {X 99.271,Y 110.691,Z 71.172,A 180.000,B 0.000,C 180.000} C_DIS
LIN {X 99.650,Y 110.644,Z 71.158,A 180.000,B 0.000,C 180.000} C_DIS
LIN {X 99.725,Y 110.633,Z 71.156,A 180.000,B 0.000,C 180.000} C_DIS
LIN {X 99.801,Y 110.620,Z 71.153,A 180.000,B 0.000,C 180.000} C_DIS
LIN {X 99.878,Y 110.607,Z 71.150,A 180.000,B 0.000,C 180.000} C_DIS
LIN {X 100.342,Y 110.522,Z 71.134,A 180.000,B 0.000,C 180.000} C_DIS
LIN {X 100.415,Y 110.509,Z 71.131,A 180.000,B 0.000,C 180.000} C_DIS
LIN {X 100.489,Y 110.494,Z 71.129,A 180.000,B 0.000,C 180.000} C_DIS
LIN {X 100.561,Y 110.477,Z 71.126,A 180.000,B 0.000,C 180.000} C_DIS
LIN {X 100.710,Y 110.441,Z 71.121,A 180.000,B 0.000,C 180.000} C_DIS
LIN {X 101.089,Y 110.350,Z 71.107,A 180.000,B 0.000,C 180.000} C_DIS
LIN {X 101.163,Y 110.332,Z 71.104,A 180.000,B 0.000,C 180.000} C_DIS
LIN {X 101.237,Y 110.312,Z 71.102,A 180.000,B 0.000,C 180.000} C_DIS
LIN {X 101.311,Y 110.289,Z 71.099,A 180.000,B 0.000,C 180.000} C_DIS
LIN {X 101.754,Y 110.156,Z 71.083,A 180.000,B 0.000,C 180.000} C_DIS
LIN {X 101.828,Y 110.134,Z 71.080,A 180.000,B 0.000,C 180.000} C_DIS
LIN {X 101.901,Y 110.111,Z 71.077,A 180.000,B 0.000,C 180.000} C_DIS
LIN {X 101.974,Y 110.087,Z 71.075,A 180.000,B 0.000,C 180.000} C_DIS
LIN {X 102.045,Y 110.061,Z 71.072,A 180.000,B 0.000,C 180.000} C_DIS
LIN {X 102.414,Y 109.927,Z 71.058,A 180.000,B 0.000,C 180.000} C_DIS
LIN {X 102.485,Y 109.901,Z 71.056,A 180.000,B 0.000,C 180.000} C_DIS
LIN {X 102.556,Y 109.875,Z 71.053,A 180.000,B 0.000,C 180.000} C_DIS
LIN {X 102.626,Y 109.848,Z 71.051,A 180.000,B 0.000,C 180.000} C_DIS
LIN {X 102.696,Y 109.819,Z 71.048,A 180.000,B 0.000,C 180.000} C_DIS
LIN {X 103.198,Y 109.604,Z 71.029,A 180.000,B 0.000,C 180.000} C_DIS
LIN {X 103.269,Y 109.573,Z 71.026,A 180.000,B 0.000,C 180.000} C_DIS
LIN {X 103.339,Y 109.541,Z 71.023,A 180.000,B 0.000,C 180.000} C_DIS
LIN {X 103.408,Y 109.508,Z 71.021,A 180.000,B 0.000,C 180.000} C_DIS
LIN {X 103.894,Y 109.266,Z 71.002,A 180.000,B 0.000,C 180.000} C_DIS
LIN {X 103.962,Y 109.232,Z 70.999,A 180.000,B 0.000,C 180.000} C_DIS
LIN {X 104.028,Y 109.196,Z 70.997,A 180.000,B 0.000,C 180.000} C_DIS
LIN {X 104.094,Y 109.159,Z 70.994,A 180.000,B 0.000,C 180.000} C_DIS
LIN {X 104.502,Y 108.927,Z 70.978,A 180.000,B 0.000,C 180.000} C_DIS
LIN {X 104.569,Y 108.889,Z 70.975,A 180.000,B 0.000,C 180.000} C_DIS
LIN {X 104.635,Y 108.849,Z 70.972,A 180.000,B 0.000,C 180.000} C_DIS
LIN {X 104.701,Y 108.809,Z 70.969,A 180.000,B 0.000,C 180.000} C_DIS
LIN {X 104.766,Y 108.767,Z 70.967,A 180.000,B 0.000,C 180.000} C_DIS
LIN {X 105.160,Y 108.512,Z 70.950,A 180.000,B 0.000,C 180.000} C_DIS
LIN {X 105.224,Y 108.471,Z 70.948,A 180.000,B 0.000,C 180.000} C_DIS
LIN {X 105.287,Y 108.429,Z 70.945,A 180.000,B 0.000,C 180.000} C_DIS
LIN {X 105.349,Y 108.384,Z 70.942,A 180.000,B 0.000,C 180.000} C_DIS
LIN {X 105.665,Y 108.154,Z 70.929,A 180.000,B 0.000,C 180.000} C_DIS
LIN {X 105.788,Y 108.065,Z 70.923,A 180.000,B 0.000,C 180.000} C_DIS
LIN {X 105.849,Y 108.020,Z 70.921,A 180.000,B 0.000,C 180.000} C_DIS
LIN {X 105.909,Y 107.972,Z 70.918,A 180.000,B 0.000,C 180.000} C_DIS
LIN {X 105.970,Y 107.923,Z 70.915,A 180.000,B 0.000,C 180.000} C_DIS
LIN {X 106.397,Y 107.575,Z 70.896,A 180.000,B 0.000,C 180.000} C_DIS
LIN {X 106.455,Y 107.526,Z 70.893,A 180.000,B 0.000,C 180.000} C_DIS
LIN {X 106.512,Y 107.475,Z 70.891,A 180.000,B 0.000,C 180.000} C_DIS
LIN {X 106.625,Y 107.373,Z 70.885,A 180.000,B 0.000,C 180.000} C_DIS
LIN {X 106.799,Y 107.213,Z 70.877,A 180.000,B 0.000,C 180.000} C_DIS
LIN {X 106.914,Y 107.108,Z 70.872,A 180.000,B 0.000,C 180.000} C_DIS
LIN {X 106.970,Y 107.057,Z 70.869,A 180.000,B 0.000,C 180.000} C_DIS
LIN {X 107.025,Y 107.004,Z 70.866,A 180.000,B 0.000,C 180.000} C_DIS
LIN {X 107.079,Y 106.949,Z 70.864,A 180.000,B 0.000,C 180.000} C_DIS
LIN {X 107.244,Y 106.780,Z 70.856,A 180.000,B 0.000,C 180.000} C_DIS
LIN {X 107.353,Y 106.668,Z 70.850,A 180.000,B 0.000,C 180.000} C_DIS
LIN {X 107.462,Y 106.557,Z 70.845,A 180.000,B 0.000,C 180.000} C_DIS
LIN {X 107.517,Y 106.501,Z 70.842,A 180.000,B 0.000,C 180.000} C_DIS
LIN {X 107.569,Y 106.444,Z 70.839,A 180.000,B 0.000,C 180.000} C_DIS
LIN {X 107.620,Y 106.386,Z 70.837,A 180.000,B 0.000,C 180.000} C_DIS
LIN {X 107.929,Y 106.033,Z 70.820,A 180.000,B 0.000,C 180.000} C_DIS
LIN {X 107.980,Y 105.975,Z 70.817,A 180.000,B 0.000,C 180.000} C_DIS
LIN {X 108.030,Y 105.916,Z 70.815,A 180.000,B 0.000,C 180.000} C_DIS
LIN {X 108.078,Y 105.856,Z 70.812,A 180.000,B 0.000,C 180.000} C_DIS
LIN {X 108.125,Y 105.796,Z 70.809,A 180.000,B 0.000,C 180.000} C_DIS
LIN {X 108.222,Y 105.672,Z 70.804,A 180.000,B 0.000,C 180.000} C_DIS
LIN {X 108.414,Y 105.424,Z 70.793,A 180.000,B 0.000,C 180.000} C_DIS
LIN {X 108.462,Y 105.363,Z 70.790,A 180.000,B 0.000,C 180.000} C_DIS
LIN {X 108.508,Y 105.301,Z 70.788,A 180.000,B 0.000,C 180.000} C_DIS
LIN {X 108.554,Y 105.237,Z 70.785,A 180.000,B 0.000,C 180.000} C_DIS
LIN {X 108.642,Y 105.110,Z 70.779,A 180.000,B 0.000,C 180.000} C_DIS
LIN {X 108.687,Y 105.046,Z 70.777,A 180.000,B 0.000,C 180.000} C_DIS
LIN {X 108.776,Y 104.916,Z 70.771,A 180.000,B 0.000,C 180.000} C_DIS
LIN {X 108.866,Y 104.787,Z 70.766,A 180.000,B 0.000,C 180.000} C_DIS
LIN {X 108.909,Y 104.723,Z 70.763,A 180.000,B 0.000,C 180.000} C_DIS
LIN {X 108.952,Y 104.659,Z 70.760,A 180.000,B 0.000,C 180.000} C_DIS
LIN {X 108.992,Y 104.593,Z 70.758,A 180.000,B 0.000,C 180.000} C_DIS
LIN {X 109.033,Y 104.527,Z 70.755,A 180.000,B 0.000,C 180.000} C_DIS
LIN {X 109.115,Y 104.393,Z 70.749,A 180.000,B 0.000,C 180.000} C_DIS
LIN {X 109.237,Y 104.193,Z 70.741,A 180.000,B 0.000,C 180.000} C_DIS
LIN {X 109.278,Y 104.127,Z 70.739,A 180.000,B 0.000,C 180.000} C_DIS
LIN {X 109.317,Y 104.060,Z 70.736,A 180.000,B 0.000,C 180.000} C_DIS
LIN {X 109.355,Y 103.993,Z 70.733,A 180.000,B 0.000,C 180.000} C_DIS
LIN {X 109.393,Y 103.924,Z 70.730,A 180.000,B 0.000,C 180.000} C_DIS
LIN {X 109.467,Y 103.785,Z 70.725,A 180.000,B 0.000,C 180.000} C_DIS
LIN {X 109.505,Y 103.716,Z 70.722,A 180.000,B 0.000,C 180.000} C_DIS
LIN {X 109.579,Y 103.578,Z 70.717,A 180.000,B 0.000,C 180.000} C_DIS
LIN {X 109.654,Y 103.439,Z 70.711,A 180.000,B 0.000,C 180.000} C_DIS
LIN {X 109.690,Y 103.370,Z 70.708,A 180.000,B 0.000,C 180.000} C_DIS
LIN {X 109.723,Y 103.301,Z 70.706,A 180.000,B 0.000,C 180.000} C_DIS
LIN {X 109.789,Y 103.160,Z 70.700,A 180.000,B 0.000,C 180.000} C_DIS
LIN {X 109.856,Y 103.017,Z 70.695,A 180.000,B 0.000,C 180.000} C_DIS
LIN {X 109.922,Y 102.875,Z 70.689,A 180.000,B 0.000,C 180.000} C_DIS
LIN {X 109.955,Y 102.804,Z 70.687,A 180.000,B 0.000,C 180.000} C_DIS
LIN {X 109.988,Y 102.734,Z 70.684,A 180.000,B 0.000,C 180.000} C_DIS
LIN {X 110.019,Y 102.662,Z 70.681,A 180.000,B 0.000,C 180.000} C_DIS
LIN {X 110.048,Y 102.590,Z 70.679,A 180.000,B 0.000,C 180.000} C_DIS
LIN {X 110.078,Y 102.518,Z 70.676,A 180.000,B 0.000,C 180.000} C_DIS
LIN {X 110.107,Y 102.445,Z 70.673,A 180.000,B 0.000,C 180.000} C_DIS
LIN {X 110.136,Y 102.372,Z 70.671,A 180.000,B 0.000,C 180.000} C_DIS
LIN {X 110.165,Y 102.299,Z 70.668,A 180.000,B 0.000,C 180.000} C_DIS
LIN {X 110.194,Y 102.226,Z 70.666,A 180.000,B 0.000,C 180.000} C_DIS
LIN {X 110.223,Y 102.153,Z 70.663,A 180.000,B 0.000,C 180.000} C_DIS
LIN {X 110.252,Y 102.081,Z 70.660,A 180.000,B 0.000,C 180.000} C_DIS
LIN {X 110.281,Y 102.008,Z 70.658,A 180.000,B 0.000,C 180.000} C_DIS
LIN {X 110.308,Y 101.935,Z 70.655,A 180.000,B 0.000,C 180.000} C_DIS
LIN {X 110.333,Y 101.860,Z 70.653,A 180.000,B 0.000,C 180.000} C_DIS
LIN {X 110.383,Y 101.712,Z 70.648,A 180.000,B 0.000,C 180.000} C_DIS
LIN {X 110.433,Y 101.563,Z 70.643,A 180.000,B 0.000,C 180.000} C_DIS
LIN {X 110.483,Y 101.413,Z 70.638,A 180.000,B 0.000,C 180.000} C_DIS
LIN {X 110.531,Y 101.265,Z 70.633,A 180.000,B 0.000,C 180.000} C_DIS
LIN {X 110.573,Y 101.115,Z 70.628,A 180.000,B 0.000,C 180.000} C_DIS
LIN {X 110.615,Y 100.963,Z 70.624,A 180.000,B 0.000,C 180.000} C_DIS
LIN {X 110.656,Y 100.811,Z 70.619,A 180.000,B 0.000,C 180.000} C_DIS
LIN {X 110.697,Y 100.660,Z 70.615,A 180.000,B 0.000,C 180.000} C_DIS
LIN {X 110.738,Y 100.508,Z 70.610,A 180.000,B 0.000,C 180.000} C_DIS
LIN {X 110.771,Y 100.355,Z 70.606,A 180.000,B 0.000,C 180.000} C_DIS
LIN {X 110.804,Y 100.202,Z 70.601,A 180.000,B 0.000,C 180.000} C_DIS
LIN {X 110.836,Y 100.048,Z 70.597,A 180.000,B 0.000,C 180.000} C_DIS
LIN {X 110.869,Y 99.894,Z 70.593,A 180.000,B 0.000,C 180.000} C_DIS
LIN {X 110.899,Y 99.740,Z 70.589,A 180.000,B 0.000,C 180.000} C_DIS
LIN {X 110.923,Y 99.586,Z 70.585,A 180.000,B 0.000,C 180.000} C_DIS
LIN {X 110.947,Y 99.430,Z 70.581,A 180.000,B 0.000,C 180.000} C_DIS
LIN {X 110.970,Y 99.274,Z 70.577,A 180.000,B 0.000,C 180.000} C_DIS
LIN {X 110.994,Y 99.119,Z 70.573,A 180.000,B 0.000,C 180.000} C_DIS
LIN {X 111.015,Y 98.964,Z 70.570,A 180.000,B 0.000,C 180.000} C_DIS
LIN {X 111.030,Y 98.807,Z 70.566,A 180.000,B 0.000,C 180.000} C_DIS
LIN {X 111.045,Y 98.651,Z 70.562,A 180.000,B 0.000,C 180.000} C_DIS
LIN {X 111.059,Y 98.494,Z 70.559,A 180.000,B 0.000,C 180.000} C_DIS
LIN {X 111.074,Y 98.337,Z 70.556,A 180.000,B 0.000,C 180.000} C_DIS
LIN {X 111.084,Y 98.181,Z 70.552,A 180.000,B 0.000,C 180.000} C_DIS
LIN {X 111.090,Y 98.024,Z 70.549,A 180.000,B 0.000,C 180.000} C_DIS
LIN {X 111.096,Y 97.867,Z 70.546,A 180.000,B 0.000,C 180.000} C_DIS
LIN {X 111.102,Y 97.709,Z 70.543,A 180.000,B 0.000,C 180.000} C_DIS
LIN {X 111.107,Y 97.552,Z 70.540,A 180.000,B 0.000,C 180.000} C_DIS
LIN {X 111.107,Y 97.395,Z 70.537,A 180.000,B 0.000,C 180.000} C_DIS
LIN {X 111.104,Y 97.238,Z 70.534,A 180.000,B 0.000,C 180.000} C_DIS
LIN {X 111.101,Y 97.080,Z 70.532,A 180.000,B 0.000,C 180.000} C_DIS
LIN {X 111.098,Y 96.923,Z 70.529,A 180.000,B 0.000,C 180.000} C_DIS
LIN {X 111.094,Y 96.765,Z 70.527,A 180.000,B 0.000,C 180.000} C_DIS
LIN {X 111.072,Y 96.452,Z 70.522,A 180.000,B 0.000,C 180.000} C_DIS
LIN {X 111.047,Y 96.138,Z 70.518,A 180.000,B 0.000,C 180.000} C_DIS
LIN {X 111.014,Y 95.825,Z 70.514,A 180.000,B 0.000,C 180.000} C_DIS
LIN {X 110.971,Y 95.513,Z 70.511,A 180.000,B 0.000,C 180.000} C_DIS
LIN {X 110.928,Y 95.201,Z 70.508,A 180.000,B 0.000,C 180.000} C_DIS
LIN {X 110.868,Y 94.892,Z 70.505,A 180.000,B 0.000,C 180.000} C_DIS
LIN {X 110.807,Y 94.583,Z 70.503,A 180.000,B 0.000,C 180.000} C_DIS
LIN {X 110.735,Y 94.276,Z 70.502,A 180.000,B 0.000,C 180.000} C_DIS
LIN {X 110.657,Y 93.971,Z 70.501,A 180.000,B 0.000,C 180.000} C_DIS
LIN {X 110.576,Y 93.667,Z 70.500,A 180.000,B 0.000,C 180.000} C_DIS
LIN {X 110.502,Y 93.434,Z 70.500,A 180.000,B 0.000,C 180.000} C_DIS
; Cutting Move Starts
LIN {X 110.409,Y 93.142,Z 70.500,A 180.000,B 0.000,C 180.000} C_DIS
LIN {X 110.349,Y 92.964,Z 70.500,A 180.000,B 0.000,C 180.000} C_DIS
LIN {X 110.304,Y 92.846,Z 70.500,A 180.000,B 0.000,C 180.000} C_DIS
LIN {X 110.126,Y 92.378,Z 70.500,A 180.000,B 0.000,C 180.000} C_DIS
LIN {X 110.074,Y 92.249,Z 70.500,A 180.000,B 0.000,C 180.000} C_DIS
LIN {X 109.994,Y 92.070,Z 70.500,A 180.000,B 0.000,C 180.000} C_DIS
LIN {X 109.834,Y 91.712,Z 70.500,A 180.000,B 0.000,C 180.000} C_DIS
LIN {X 109.768,Y 91.569,Z 70.500,A 180.000,B 0.000,C 180.000} C_DIS
LIN {X 109.750,Y 91.533,Z 70.500,A 180.000,B 0.000,C 180.000} C_DIS
LIN {X 109.566,Y 91.176,Z 70.500,A 180.000,B 0.000,C 180.000} C_DIS
LIN {X 109.473,Y 90.997,Z 70.500,A 180.000,B 0.000,C 180.000} C_DIS
LIN {X 109.410,Y 90.881,Z 70.500,A 180.000,B 0.000,C 180.000} C_DIS
LIN {X 109.374,Y 90.818,Z 70.500,A 180.000,B 0.000,C 180.000} C_DIS
LIN {X 109.163,Y 90.461,Z 70.500,A 180.000,B 0.000,C 180.000} C_DIS
LIN {X 109.058,Y 90.282,Z 70.500,A 180.000,B 0.000,C 180.000} C_DIS
LIN {X 109.053,Y 90.274,Z 70.500,A 180.000,B 0.000,C 180.000} C_DIS
LIN {X 108.941,Y 90.103,Z 70.500,A 180.000,B 0.000,C 180.000} C_DIS
LIN {X 108.695,Y 89.735,Z 70.500,A 180.000,B 0.000,C 180.000} C_DIS
LIN {X 108.578,Y 89.567,Z 70.500,A 180.000,B 0.000,C 180.000} C_DIS
LIN {X 108.517,Y 89.485,Z 70.500,A 180.000,B 0.000,C 180.000} C_DIS
LIN {X 108.309,Y 89.209,Z 70.500,A 180.000,B 0.000,C 180.000} C_DIS
LIN {X 108.175,Y 89.031,Z 70.500,A 180.000,B 0.000,C 180.000} C_DIS
LIN {X 108.159,Y 89.011,Z 70.500,A 180.000,B 0.000,C 180.000} C_DIS
LIN {X 108.027,Y 88.852,Z 70.500,A 180.000,B 0.000,C 180.000} C_DIS
LIN {X 107.725,Y 88.494,Z 70.500,A 180.000,B 0.000,C 180.000} C_DIS
LIN {X 107.623,Y 88.379,Z 70.500,A 180.000,B 0.000,C 180.000} C_DIS
LIN {X 107.563,Y 88.316,Z 70.500,A 180.000,B 0.000,C 180.000} C_DIS
LIN {X 107.225,Y 87.958,Z 70.500,A 180.000,B 0.000,C 180.000} C_DIS
LIN {X 107.086,Y 87.817,Z 70.500,A 180.000,B 0.000,C 180.000} C_DIS
LIN {X 107.047,Y 87.779,Z 70.500,A 180.000,B 0.000,C 180.000} C_DIS
LIN {X 106.669,Y 87.422,Z 70.500,A 180.000,B 0.000,C 180.000} C_DIS
LIN {X 106.550,Y 87.313,Z 70.500,A 180.000,B 0.000,C 180.000} C_DIS
LIN {X 106.467,Y 87.243,Z 70.500,A 180.000,B 0.000,C 180.000} C_DIS
LIN {X 106.193,Y 87.011,Z 70.500,A 180.000,B 0.000,C 180.000} C_DIS
LIN {X 106.043,Y 86.885,Z 70.500,A 180.000,B 0.000,C 180.000} C_DIS
LIN {X 106.014,Y 86.861,Z 70.500,A 180.000,B 0.000,C 180.000} C_DIS
LIN {X 105.835,Y 86.724,Z 70.500,A 180.000,B 0.000,C 180.000} C_DIS
LIN {X 105.477,Y 86.455,Z 70.500,A 180.000,B 0.000,C 180.000} C_DIS
LIN {X 105.331,Y 86.349,Z 70.500,A 180.000,B 0.000,C 180.000} C_DIS
LIN {X 104.941,Y 86.089,Z 70.500,A 180.000,B 0.000,C 180.000} C_DIS
LIN {X 104.795,Y 85.992,Z 70.500,A 180.000,B 0.000,C 180.000} C_DIS
LIN {X 104.762,Y 85.971,Z 70.500,A 180.000,B 0.000,C 180.000} C_DIS
LIN {X 104.584,Y 85.863,Z 70.500,A 180.000,B 0.000,C 180.000} C_DIS
LIN {X 104.196,Y 85.634,Z 70.500,A 180.000,B 0.000,C 180.000} C_DIS
LIN {X 104.047,Y 85.550,Z 70.500,A 180.000,B 0.000,C 180.000} C_DIS
LIN {X 103.865,Y 85.455,Z 70.500,A 180.000,B 0.000,C 180.000} C_DIS
LIN {X 103.511,Y 85.273,Z 70.500,A 180.000,B 0.000,C 180.000} C_DIS
LIN {X 103.332,Y 85.186,Z 70.500,A 180.000,B 0.000,C 180.000} C_DIS
LIN {X 102.975,Y 85.026,Z 70.500,A 180.000,B 0.000,C 180.000} C_DIS
LIN {X 102.796,Y 84.946,Z 70.500,A 180.000,B 0.000,C 180.000} C_DIS
LIN {X 102.734,Y 84.919,Z 70.500,A 180.000,B 0.000,C 180.000} C_DIS
LIN {X 102.617,Y 84.872,Z 70.500,A 180.000,B 0.000,C 180.000} C_DIS
LIN {X 102.081,Y 84.667,Z 70.500,A 180.000,B 0.000,C 180.000} C_DIS
LIN {X 101.902,Y 84.606,Z 70.500,A 180.000,B 0.000,C 180.000} C_DIS
LIN {X 101.366,Y 84.435,Z 70.500,A 180.000,B 0.000,C 180.000} C_DIS
LIN {X 101.187,Y 84.383,Z 70.500,A 180.000,B 0.000,C 180.000} C_DIS
LIN {X 100.651,Y 84.244,Z 70.500,A 180.000,B 0.000,C 180.000} C_DIS
LIN {X 100.480,Y 84.204,Z 70.500,A 180.000,B 0.000,C 180.000} C_DIS
LIN {X 100.472,Y 84.202,Z 70.500,A 180.000,B 0.000,C 180.000} C_DIS
LIN {X 99.936,Y 84.096,Z 70.500,A 180.000,B 0.000,C 180.000} C_DIS
LIN {X 99.757,Y 84.062,Z 70.500,A 180.000,B 0.000,C 180.000} C_DIS
LIN {X 99.578,Y 84.036,Z 70.500,A 180.000,B 0.000,C 180.000} C_DIS
LIN {X 99.221,Y 83.985,Z 70.500,A 180.000,B 0.000,C 180.000} C_DIS
LIN {X 99.042,Y 83.961,Z 70.500,A 180.000,B 0.000,C 180.000} C_DIS
LIN {X 98.863,Y 83.944,Z 70.500,A 180.000,B 0.000,C 180.000} C_DIS
LIN {X 98.505,Y 83.914,Z 70.500,A 180.000,B 0.000,C 180.000} C_DIS
LIN {X 98.327,Y 83.899,Z 70.500,A 180.000,B 0.000,C 180.000} C_DIS
LIN {X 98.148,Y 83.891,Z 70.500,A 180.000,B 0.000,C 180.000} C_DIS
LIN {X 97.612,Y 83.875,Z 70.500,A 180.000,B 0.000,C 180.000} C_DIS
LIN {X 97.433,Y 83.874,Z 70.500,A 180.000,B 0.000,C 180.000} C_DIS
LIN {X 96.897,Y 83.889,Z 70.500,A 180.000,B 0.000,C 180.000} C_DIS
LIN {X 96.718,Y 83.897,Z 70.500,A 180.000,B 0.000,C 180.000} C_DIS
LIN {X 96.539,Y 83.911,Z 70.500,A 180.000,B 0.000,C 180.000} C_DIS
LIN {X 96.181,Y 83.941,Z 70.500,A 180.000,B 0.000,C 180.000} C_DIS
LIN {X 96.003,Y 83.956,Z 70.500,A 180.000,B 0.000,C 180.000} C_DIS
LIN {X 95.824,Y 83.979,Z 70.500,A 180.000,B 0.000,C 180.000} C_DIS
LIN {X 95.466,Y 84.030,Z 70.500,A 180.000,B 0.000,C 180.000} C_DIS
LIN {X 95.288,Y 84.055,Z 70.500,A 180.000,B 0.000,C 180.000} C_DIS
LIN {X 95.109,Y 84.087,Z 70.500,A 180.000,B 0.000,C 180.000} C_DIS
LIN {X 94.573,Y 84.194,Z 70.500,A 180.000,B 0.000,C 180.000} C_DIS
LIN {X 94.520,Y 84.204,Z 70.500,A 180.000,B 0.000,C 180.000} C_DIS
LIN {X 94.394,Y 84.233,Z 70.500,A 180.000,B 0.000,C 180.000} C_DIS
LIN {X 93.813,Y 84.383,Z 70.500,A 180.000,B 0.000,C 180.000} C_DIS
LIN {X 93.679,Y 84.421,Z 70.500,A 180.000,B 0.000,C 180.000} C_DIS
LIN {X 93.500,Y 84.478,Z 70.500,A 180.000,B 0.000,C 180.000} C_DIS
LIN {X 93.142,Y 84.592,Z 70.500,A 180.000,B 0.000,C 180.000} C_DIS
LIN {X 92.964,Y 84.651,Z 70.500,A 180.000,B 0.000,C 180.000} C_DIS
LIN {X 92.785,Y 84.719,Z 70.500,A 180.000,B 0.000,C 180.000} C_DIS
LIN {X 92.427,Y 84.855,Z 70.500,A 180.000,B 0.000,C 180.000} C_DIS
LIN {X 92.266,Y 84.919,Z 70.500,A 180.000,B 0.000,C 180.000} C_DIS
LIN {X 92.249,Y 84.926,Z 70.500,A 180.000,B 0.000,C 180.000} C_DIS
LIN {X 92.070,Y 85.006,Z 70.500,A 180.000,B 0.000,C 180.000} C_DIS
LIN {X 91.712,Y 85.166,Z 70.500,A 180.000,B 0.000,C 180.000} C_DIS
LIN {X 91.533,Y 85.250,Z 70.500,A 180.000,B 0.000,C 180.000} C_DIS
LIN {X 91.481,Y 85.276,Z 70.500,A 180.000,B 0.000,C 180.000} C_DIS
LIN {X 90.997,Y 85.527,Z 70.500,A 180.000,B 0.000,C 180.000} C_DIS
LIN {X 90.818,Y 85.626,Z 70.500,A 180.000,B 0.000,C 180.000} C_DIS
LIN {X 90.461,Y 85.837,Z 70.500,A 180.000,B 0.000,C 180.000} C_DIS
LIN {X 90.282,Y 85.943,Z 70.500,A 180.000,B 0.000,C 180.000} C_DIS
LIN {X 90.205,Y 85.992,Z 70.500,A 180.000,B 0.000,C 180.000} C_DIS
LIN {X 90.103,Y 86.059,Z 70.500,A 180.000,B 0.000,C 180.000} C_DIS
LIN {X 89.669,Y 86.349,Z 70.500,A 180.000,B 0.000,C 180.000} C_DIS
LIN {X 89.567,Y 86.421,Z 70.500,A 180.000,B 0.000,C 180.000} C_DIS
LIN {X 89.425,Y 86.528,Z 70.500,A 180.000,B 0.000,C 180.000} C_DIS
LIN {X 89.188,Y 86.707,Z 70.500,A 180.000,B 0.000,C 180.000} C_DIS
LIN {X 89.031,Y 86.825,Z 70.500,A 180.000,B 0.000,C 180.000} C_DIS
LIN {X 88.957,Y 86.885,Z 70.500,A 180.000,B 0.000,C 180.000} C_DIS
LIN {X 88.852,Y 86.974,Z 70.500,A 180.000,B 0.000,C 180.000} C_DIS
LIN {X 88.494,Y 87.276,Z 70.500,A 180.000,B 0.000,C 180.000} C_DIS
LIN {X 88.331,Y 87.422,Z 70.500,A 180.000,B 0.000,C 180.000} C_DIS
LIN {X 87.953,Y 87.779,Z 70.500,A 180.000,B 0.000,C 180.000} C_DIS
LIN {X 87.779,Y 87.954,Z 70.500,A 180.000,B 0.000,C 180.000} C_DIS
LIN {X 87.422,Y 88.332,Z 70.500,A 180.000,B 0.000,C 180.000} C_DIS
LIN {X 87.275,Y 88.494,Z 70.500,A 180.000,B 0.000,C 180.000} C_DIS
LIN {X 86.973,Y 88.852,Z 70.500,A 180.000,B 0.000,C 180.000} C_DIS
LIN {X 86.885,Y 88.956,Z 70.500,A 180.000,B 0.000,C 180.000} C_DIS
LIN {X 86.825,Y 89.031,Z 70.500,A 180.000,B 0.000,C 180.000} C_DIS
LIN {X 86.707,Y 89.188,Z 70.500,A 180.000,B 0.000,C 180.000} C_DIS
LIN {X 86.528,Y 89.426,Z 70.500,A 180.000,B 0.000,C 180.000} C_DIS
LIN {X 86.422,Y 89.567,Z 70.500,A 180.000,B 0.000,C 180.000} C_DIS
LIN {X 86.349,Y 89.669,Z 70.500,A 180.000,B 0.000,C 180.000} C_DIS
LIN {X 86.298,Y 89.746,Z 70.500,A 180.000,B 0.000,C 180.000} C_DIS
LIN {X 86.059,Y 90.103,Z 70.500,A 180.000,B 0.000,C 180.000} C_DIS
LIN {X 85.992,Y 90.204,Z 70.500,A 180.000,B 0.000,C 180.000} C_DIS
LIN {X 85.942,Y 90.282,Z 70.500,A 180.000,B 0.000,C 180.000} C_DIS
LIN {X 85.837,Y 90.461,Z 70.500,A 180.000,B 0.000,C 180.000} C_DIS
LIN {X 85.626,Y 90.818,Z 70.500,A 180.000,B 0.000,C 180.000} C_DIS
LIN {X 85.527,Y 90.997,Z 70.500,A 180.000,B 0.000,C 180.000} C_DIS
LIN {X 85.276,Y 91.482,Z 70.500,A 180.000,B 0.000,C 180.000} C_DIS
LIN {X 85.250,Y 91.533,Z 70.500,A 180.000,B 0.000,C 180.000} C_DIS
LIN {X 85.166,Y 91.712,Z 70.500,A 180.000,B 0.000,C 180.000} C_DIS
LIN {X 85.006,Y 92.070,Z 70.500,A 180.000,B 0.000,C 180.000} C_DIS
LIN {X 84.926,Y 92.249,Z 70.500,A 180.000,B 0.000,C 180.000} C_DIS
LIN {X 84.919,Y 92.266,Z 70.500,A 180.000,B 0.000,C 180.000} C_DIS
LIN {X 84.856,Y 92.427,Z 70.500,A 180.000,B 0.000,C 180.000} C_DIS
LIN {X 84.719,Y 92.785,Z 70.500,A 180.000,B 0.000,C 180.000} C_DIS
LIN {X 84.651,Y 92.964,Z 70.500,A 180.000,B 0.000,C 180.000} C_DIS
LIN {X 84.591,Y 93.142,Z 70.500,A 180.000,B 0.000,C 180.000} C_DIS
LIN {X 84.477,Y 93.500,Z 70.500,A 180.000,B 0.000,C 180.000} C_DIS
LIN {X 84.421,Y 93.679,Z 70.500,A 180.000,B 0.000,C 180.000} C_DIS
LIN {X 84.383,Y 93.816,Z 70.500,A 180.000,B 0.000,C 180.000} C_DIS
LIN {X 84.280,Y 94.215,Z 70.500,A 180.000,B 0.000,C 180.000} C_DIS
LIN {X 84.234,Y 94.394,Z 70.500,A 180.000,B 0.000,C 180.000} C_DIS
LIN {X 84.204,Y 94.519,Z 70.500,A 180.000,B 0.000,C 180.000} C_DIS
LIN {X 84.193,Y 94.573,Z 70.500,A 180.000,B 0.000,C 180.000} C_DIS
LIN {X 84.086,Y 95.109,Z 70.500,A 180.000,B 0.000,C 180.000} C_DIS
LIN {X 84.055,Y 95.288,Z 70.500,A 180.000,B 0.000,C 180.000} C_DIS
LIN {X 83.979,Y 95.824,Z 70.500,A 180.000,B 0.000,C 180.000} C_DIS
LIN {X 83.956,Y 96.003,Z 70.500,A 180.000,B 0.000,C 180.000} C_DIS
LIN {X 83.940,Y 96.181,Z 70.500,A 180.000,B 0.000,C 180.000} C_DIS
LIN {X 83.910,Y 96.539,Z 70.500,A 180.000,B 0.000,C 180.000} C_DIS
LIN {X 83.896,Y 96.718,Z 70.500,A 180.000,B 0.000,C 180.000} C_DIS
LIN {X 83.889,Y 96.897,Z 70.500,A 180.000,B 0.000,C 180.000} C_DIS
LIN {X 83.879,Y 97.254,Z 70.500,A 180.000,B 0.000,C 180.000} C_DIS
LIN {X 83.874,Y 97.433,Z 70.500,A 180.000,B 0.000,C 180.000} C_DIS
LIN {X 83.876,Y 97.612,Z 70.500,A 180.000,B 0.000,C 180.000} C_DIS
LIN {X 83.891,Y 98.148,Z 70.500,A 180.000,B 0.000,C 180.000} C_DIS
LIN {X 83.899,Y 98.327,Z 70.500,A 180.000,B 0.000,C 180.000} C_DIS
LIN {X 83.914,Y 98.505,Z 70.500,A 180.000,B 0.000,C 180.000} C_DIS
LIN {X 83.944,Y 98.863,Z 70.500,A 180.000,B 0.000,C 180.000} C_DIS
LIN {X 83.961,Y 99.042,Z 70.500,A 180.000,B 0.000,C 180.000} C_DIS
LIN {X 83.986,Y 99.221,Z 70.500,A 180.000,B 0.000,C 180.000} C_DIS
LIN {X 84.036,Y 99.578,Z 70.500,A 180.000,B 0.000,C 180.000} C_DIS
LIN {X 84.062,Y 99.757,Z 70.500,A 180.000,B 0.000,C 180.000} C_DIS
LIN {X 84.095,Y 99.936,Z 70.500,A 180.000,B 0.000,C 180.000} C_DIS
LIN {X 84.166,Y 100.293,Z 70.500,A 180.000,B 0.000,C 180.000} C_DIS
LIN {X 84.202,Y 100.472,Z 70.500,A 180.000,B 0.000,C 180.000} C_DIS
LIN {X 84.204,Y 100.481,Z 70.500,A 180.000,B 0.000,C 180.000} C_DIS
LIN {X 84.245,Y 100.651,Z 70.500,A 180.000,B 0.000,C 180.000} C_DIS
LIN {X 84.383,Y 101.187,Z 70.500,A 180.000,B 0.000,C 180.000} C_DIS
LIN {X 84.434,Y 101.366,Z 70.500,A 180.000,B 0.000,C 180.000} C_DIS
LIN {X 84.605,Y 101.902,Z 70.500,A 180.000,B 0.000,C 180.000} C_DIS
LIN {X 84.668,Y 102.081,Z 70.500,A 180.000,B 0.000,C 180.000} C_DIS
LIN {X 84.873,Y 102.617,Z 70.500,A 180.000,B 0.000,C 180.000} C_DIS
LIN {X 84.919,Y 102.734,Z 70.500,A 180.000,B 0.000,C 180.000} C_DIS
LIN {X 84.946,Y 102.796,Z 70.500,A 180.000,B 0.000,C 180.000} C_DIS
LIN {X 85.186,Y 103.332,Z 70.500,A 180.000,B 0.000,C 180.000} C_DIS
LIN {X 85.273,Y 103.511,Z 70.500,A 180.000,B 0.000,C 180.000} C_DIS
LIN {X 85.457,Y 103.869,Z 70.500,A 180.000,B 0.000,C 180.000} C_DIS
LIN {X 85.550,Y 104.047,Z 70.500,A 180.000,B 0.000,C 180.000} C_DIS
LIN {X 85.634,Y 104.196,Z 70.500,A 180.000,B 0.000,C 180.000} C_DIS
LIN {X 85.863,Y 104.584,Z 70.500,A 180.000,B 0.000,C 180.000} C_DIS
LIN {X 85.970,Y 104.762,Z 70.500,A 180.000,B 0.000,C 180.000} C_DIS
LIN {X 85.992,Y 104.796,Z 70.500,A 180.000,B 0.000,C 180.000} C_DIS
LIN {X 86.089,Y 104.941,Z 70.500,A 180.000,B 0.000,C 180.000} C_DIS
LIN {X 86.327,Y 105.299,Z 70.500,A 180.000,B 0.000,C 180.000} C_DIS
LIN {X 86.349,Y 105.331,Z 70.500,A 180.000,B 0.000,C 180.000} C_DIS
LIN {X 86.455,Y 105.477,Z 70.500,A 180.000,B 0.000,C 180.000} C_DIS
LIN {X 86.724,Y 105.835,Z 70.500,A 180.000,B 0.000,C 180.000} C_DIS
LIN {X 86.860,Y 106.014,Z 70.500,A 180.000,B 0.000,C 180.000} C_DIS
LIN {X 86.885,Y 106.044,Z 70.500,A 180.000,B 0.000,C 180.000} C_DIS
LIN {X 87.011,Y 106.193,Z 70.500,A 180.000,B 0.000,C 180.000} C_DIS
LIN {X 87.243,Y 106.468,Z 70.500,A 180.000,B 0.000,C 180.000} C_DIS
LIN {X 87.313,Y 106.550,Z 70.500,A 180.000,B 0.000,C 180.000} C_DIS
LIN {X 87.422,Y 106.668,Z 70.500,A 180.000,B 0.000,C 180.000} C_DIS
LIN {X 87.817,Y 107.086,Z 70.500,A 180.000,B 0.000,C 180.000} C_DIS
LIN {X 87.958,Y 107.226,Z 70.500,A 180.000,B 0.000,C 180.000} C_DIS
LIN {X 88.316,Y 107.564,Z 70.500,A 180.000,B 0.000,C 180.000} C_DIS
LIN {X 88.378,Y 107.623,Z 70.500,A 180.000,B 0.000,C 180.000} C_DIS
LIN {X 88.494,Y 107.724,Z 70.500,A 180.000,B 0.000,C 180.000} C_DIS
LIN {X 88.852,Y 108.026,Z 70.500,A 180.000,B 0.000,C 180.000} C_DIS
LIN {X 89.011,Y 108.159,Z 70.500,A 180.000,B 0.000,C 180.000} C_DIS
LIN {X 89.031,Y 108.175,Z 70.500,A 180.000,B 0.000,C 180.000} C_DIS
LIN {X 89.209,Y 108.310,Z 70.500,A 180.000,B 0.000,C 180.000} C_DIS
LIN {X 89.484,Y 108.517,Z 70.500,A 180.000,B 0.000,C 180.000} C_DIS
LIN {X 89.567,Y 108.579,Z 70.500,A 180.000,B 0.000,C 180.000} C_DIS
LIN {X 89.736,Y 108.695,Z 70.500,A 180.000,B 0.000,C 180.000} C_DIS
LIN {X 90.103,Y 108.941,Z 70.500,A 180.000,B 0.000,C 180.000} C_DIS
LIN {X 90.275,Y 109.053,Z 70.500,A 180.000,B 0.000,C 180.000} C_DIS
LIN {X 90.282,Y 109.057,Z 70.500,A 180.000,B 0.000,C 180.000} C_DIS
LIN {X 90.461,Y 109.163,Z 70.500,A 180.000,B 0.000,C 180.000} C_DIS
LIN {X 90.818,Y 109.374,Z 70.500,A 180.000,B 0.000,C 180.000} C_DIS
LIN {X 90.880,Y 109.410,Z 70.500,A 180.000,B 0.000,C 180.000} C_DIS
LIN {X 90.997,Y 109.473,Z 70.500,A 180.000,B 0.000,C 180.000} C_DIS
LIN {X 91.355,Y 109.658,Z 70.500,A 180.000,B 0.000,C 180.000} C_DIS
LIN {X 91.533,Y 109.750,Z 70.500,A 180.000,B 0.000,C 180.000} C_DIS
LIN {X 91.570,Y 109.768,Z 70.500,A 180.000,B 0.000,C 180.000} C_DIS
LIN {X 91.712,Y 109.834,Z 70.500,A 180.000,B 0.000,C 180.000} C_DIS
LIN {X 92.070,Y 109.994,Z 70.500,A 180.000,B 0.000,C 180.000} C_DIS
LIN {X 92.249,Y 110.074,Z 70.500,A 180.000,B 0.000,C 180.000} C_DIS
LIN {X 92.377,Y 110.126,Z 70.500,A 180.000,B 0.000,C 180.000} C_DIS
LIN {X 92.845,Y 110.304,Z 70.500,A 180.000,B 0.000,C 180.000} C_DIS
LIN {X 92.964,Y 110.349,Z 70.500,A 180.000,B 0.000,C 180.000} C_DIS
LIN {X 93.142,Y 110.408,Z 70.500,A 180.000,B 0.000,C 180.000} C_DIS
LIN {X 93.500,Y 110.522,Z 70.500,A 180.000,B 0.000,C 180.000} C_DIS
LIN {X 93.679,Y 110.579,Z 70.500,A 180.000,B 0.000,C 180.000} C_DIS
LIN {X 93.857,Y 110.629,Z 70.500,A 180.000,B 0.000,C 180.000} C_DIS
LIN {X 94.394,Y 110.767,Z 70.500,A 180.000,B 0.000,C 180.000} C_DIS
LIN {X 94.573,Y 110.806,Z 70.500,A 180.000,B 0.000,C 180.000} C_DIS
LIN {X 95.109,Y 110.913,Z 70.500,A 180.000,B 0.000,C 180.000} C_DIS
LIN {X 95.288,Y 110.945,Z 70.500,A 180.000,B 0.000,C 180.000} C_DIS
LIN {X 95.466,Y 110.970,Z 70.500,A 180.000,B 0.000,C 180.000} C_DIS
LIN {X 95.824,Y 111.021,Z 70.500,A 180.000,B 0.000,C 180.000} C_DIS
LIN {X 96.003,Y 111.044,Z 70.500,A 180.000,B 0.000,C 180.000} C_DIS
LIN {X 96.181,Y 111.059,Z 70.500,A 180.000,B 0.000,C 180.000} C_DIS
LIN {X 96.539,Y 111.089,Z 70.500,A 180.000,B 0.000,C 180.000} C_DIS
LIN {X 96.718,Y 111.103,Z 70.500,A 180.000,B 0.000,C 180.000} C_DIS
LIN {X 96.897,Y 111.111,Z 70.500,A 180.000,B 0.000,C 180.000} C_DIS
LIN {X 97.433,Y 111.126,Z 70.500,A 180.000,B 0.000,C 180.000} C_DIS
LIN {X 97.612,Y 111.125,Z 70.500,A 180.000,B 0.000,C 180.000} C_DIS
LIN {X 98.148,Y 111.109,Z 70.500,A 180.000,B 0.000,C 180.000} C_DIS
LIN {X 98.327,Y 111.101,Z 70.500,A 180.000,B 0.000,C 180.000} C_DIS
LIN {X 98.505,Y 111.086,Z 70.500,A 180.000,B 0.000,C 180.000} C_DIS
LIN {X 98.863,Y 111.056,Z 70.500,A 180.000,B 0.000,C 180.000} C_DIS
LIN {X 99.042,Y 111.039,Z 70.500,A 180.000,B 0.000,C 180.000} C_DIS
LIN {X 99.187,Y 111.019,Z 70.500,A 180.000,B 0.000,C 180.000} C_DIS
LIN {X 99.578,Y 110.964,Z 70.500,A 180.000,B 0.000,C 180.000} C_DIS
LIN {X 99.757,Y 110.938,Z 70.500,A 180.000,B 0.000,C 180.000} C_DIS
LIN {X 99.936,Y 110.904,Z 70.500,A 180.000,B 0.000,C 180.000} C_DIS
LIN {X 100.472,Y 110.798,Z 70.500,A 180.000,B 0.000,C 180.000} C_DIS
LIN {X 100.651,Y 110.756,Z 70.500,A 180.000,B 0.000,C 180.000} C_DIS
LIN {X 101.187,Y 110.617,Z 70.500,A 180.000,B 0.000,C 180.000} C_DIS
LIN {X 101.366,Y 110.565,Z 70.500,A 180.000,B 0.000,C 180.000} C_DIS
LIN {X 101.902,Y 110.394,Z 70.500,A 180.000,B 0.000,C 180.000} C_DIS
LIN {X 102.081,Y 110.333,Z 70.500,A 180.000,B 0.000,C 180.000} C_DIS
LIN {X 102.623,Y 110.126,Z 70.500,A 180.000,B 0.000,C 180.000} C_DIS
LIN {X 102.796,Y 110.054,Z 70.500,A 180.000,B 0.000,C 180.000} C_DIS
LIN {X 103.153,Y 109.894,Z 70.500,A 180.000,B 0.000,C 180.000} C_DIS
LIN {X 103.332,Y 109.814,Z 70.500,A 180.000,B 0.000,C 180.000} C_DIS
LIN {X 103.430,Y 109.768,Z 70.500,A 180.000,B 0.000,C 180.000} C_DIS
LIN {X 103.511,Y 109.727,Z 70.500,A 180.000,B 0.000,C 180.000} C_DIS
LIN {X 103.869,Y 109.543,Z 70.500,A 180.000,B 0.000,C 180.000} C_DIS
LIN {X 104.047,Y 109.450,Z 70.500,A 180.000,B 0.000,C 180.000} C_DIS
LIN {X 104.120,Y 109.410,Z 70.500,A 180.000,B 0.000,C 180.000} C_DIS
LIN {X 104.226,Y 109.348,Z 70.500,A 180.000,B 0.000,C 180.000} C_DIS
LIN {X 104.584,Y 109.137,Z 70.500,A 180.000,B 0.000,C 180.000} C_DIS
LIN {X 104.725,Y 109.053,Z 70.500,A 180.000,B 0.000,C 180.000} C_DIS
LIN {X 104.762,Y 109.029,Z 70.500,A 180.000,B 0.000,C 180.000} C_DIS
LIN {X 104.941,Y 108.911,Z 70.500,A 180.000,B 0.000,C 180.000} C_DIS
LIN {X 105.299,Y 108.672,Z 70.500,A 180.000,B 0.000,C 180.000} C_DIS
LIN {X 105.477,Y 108.545,Z 70.500,A 180.000,B 0.000,C 180.000} C_DIS
LIN {X 105.835,Y 108.276,Z 70.500,A 180.000,B 0.000,C 180.000} C_DIS
LIN {X 105.989,Y 108.159,Z 70.500,A 180.000,B 0.000,C 180.000} C_DIS
LIN {X 106.014,Y 108.139,Z 70.500,A 180.000,B 0.000,C 180.000} C_DIS
LIN {X 106.193,Y 107.989,Z 70.500,A 180.000,B 0.000,C 180.000} C_DIS
LIN {X 106.414,Y 107.802,Z 70.500,A 180.000,B 0.000,C 180.000} C_DIS
LIN {X 106.550,Y 107.687,Z 70.500,A 180.000,B 0.000,C 180.000} C_DIS
LIN {X 106.622,Y 107.623,Z 70.500,A 180.000,B 0.000,C 180.000} C_DIS
LIN {X 106.729,Y 107.522,Z 70.500,A 180.000,B 0.000,C 180.000} C_DIS
LIN {X 107.000,Y 107.265,Z 70.500,A 180.000,B 0.000,C 180.000} C_DIS
LIN {X 107.086,Y 107.183,Z 70.500,A 180.000,B 0.000,C 180.000} C_DIS
LIN {X 107.183,Y 107.086,Z 70.500,A 180.000,B 0.000,C 180.000} C_DIS
LIN {X 107.521,Y 106.729,Z 70.500,A 180.000,B 0.000,C 180.000} C_DIS
LIN {X 107.623,Y 106.621,Z 70.500,A 180.000,B 0.000,C 180.000} C_DIS
LIN {X 107.687,Y 106.550,Z 70.500,A 180.000,B 0.000,C 180.000} C_DIS
LIN {X 107.802,Y 106.415,Z 70.500,A 180.000,B 0.000,C 180.000} C_DIS
LIN {X 107.989,Y 106.193,Z 70.500,A 180.000,B 0.000,C 180.000} C_DIS
LIN {X 108.140,Y 106.014,Z 70.500,A 180.000,B 0.000,C 180.000} C_DIS
LIN {X 108.159,Y 105.989,Z 70.500,A 180.000,B 0.000,C 180.000} C_DIS
LIN {X 108.276,Y 105.835,Z 70.500,A 180.000,B 0.000,C 180.000} C_DIS
LIN {X 108.545,Y 105.477,Z 70.500,A 180.000,B 0.000,C 180.000} C_DIS
LIN {X 108.673,Y 105.299,Z 70.500,A 180.000,B 0.000,C 180.000} C_DIS
LIN {X 108.911,Y 104.941,Z 70.500,A 180.000,B 0.000,C 180.000} C_DIS
LIN {X 109.030,Y 104.762,Z 70.500,A 180.000,B 0.000,C 180.000} C_DIS
LIN {X 109.053,Y 104.726,Z 70.500,A 180.000,B 0.000,C 180.000} C_DIS
LIN {X 109.137,Y 104.584,Z 70.500,A 180.000,B 0.000,C 180.000} C_DIS
LIN {X 109.348,Y 104.226,Z 70.500,A 180.000,B 0.000,C 180.000} C_DIS
LIN {X 109.410,Y 104.119,Z 70.500,A 180.000,B 0.000,C 180.000} C_DIS
LIN {X 109.450,Y 104.047,Z 70.500,A 180.000,B 0.000,C 180.000} C_DIS
LIN {X 109.543,Y 103.869,Z 70.500,A 180.000,B 0.000,C 180.000} C_DIS
LIN {X 109.727,Y 103.511,Z 70.500,A 180.000,B 0.000,C 180.000} C_DIS
LIN {X 109.768,Y 103.431,Z 70.500,A 180.000,B 0.000,C 180.000} C_DIS
LIN {X 109.814,Y 103.332,Z 70.500,A 180.000,B 0.000,C 180.000} C_DIS
LIN {X 110.054,Y 102.796,Z 70.500,A 180.000,B 0.000,C 180.000} C_DIS
LIN {X 110.126,Y 102.622,Z 70.500,A 180.000,B 0.000,C 180.000} C_DIS
LIN {X 110.332,Y 102.081,Z 70.500,A 180.000,B 0.000,C 180.000} C_DIS
LIN {X 110.395,Y 101.902,Z 70.500,A 180.000,B 0.000,C 180.000} C_DIS
LIN {X 110.566,Y 101.366,Z 70.500,A 180.000,B 0.000,C 180.000} C_DIS
LIN {X 110.617,Y 101.187,Z 70.500,A 180.000,B 0.000,C 180.000} C_DIS
LIN {X 110.755,Y 100.651,Z 70.500,A 180.000,B 0.000,C 180.000} C_DIS
LIN {X 110.798,Y 100.472,Z 70.500,A 180.000,B 0.000,C 180.000} C_DIS
LIN {X 110.834,Y 100.293,Z 70.500,A 180.000,B 0.000,C 180.000} C_DIS
LIN {X 110.905,Y 99.936,Z 70.500,A 180.000,B 0.000,C 180.000} C_DIS
LIN {X 110.938,Y 99.757,Z 70.500,A 180.000,B 0.000,C 180.000} C_DIS
LIN {X 110.964,Y 99.578,Z 70.500,A 180.000,B 0.000,C 180.000} C_DIS
LIN {X 111.019,Y 99.184,Z 70.500,A 180.000,B 0.000,C 180.000} C_DIS
LIN {X 111.039,Y 99.042,Z 70.500,A 180.000,B 0.000,C 180.000} C_DIS
LIN {X 111.056,Y 98.863,Z 70.500,A 180.000,B 0.000,C 180.000} C_DIS
LIN {X 111.086,Y 98.505,Z 70.500,A 180.000,B 0.000,C 180.000} C_DIS
LIN {X 111.101,Y 98.327,Z 70.500,A 180.000,B 0.000,C 180.000} C_DIS
LIN {X 111.109,Y 98.148,Z 70.500,A 180.000,B 0.000,C 180.000} C_DIS
LIN {X 111.124,Y 97.612,Z 70.500,A 180.000,B 0.000,C 180.000} C_DIS
LIN {X 111.126,Y 97.433,Z 70.500,A 180.000,B 0.000,C 180.000} C_DIS
LIN {X 111.121,Y 97.254,Z 70.500,A 180.000,B 0.000,C 180.000} C_DIS
LIN {X 111.111,Y 96.897,Z 70.500,A 180.000,B 0.000,C 180.000} C_DIS
LIN {X 111.104,Y 96.718,Z 70.500,A 180.000,B 0.000,C 180.000} C_DIS
LIN {X 111.090,Y 96.539,Z 70.500,A 180.000,B 0.000,C 180.000} C_DIS
LIN {X 111.060,Y 96.181,Z 70.500,A 180.000,B 0.000,C 180.000} C_DIS
LIN {X 111.044,Y 96.003,Z 70.500,A 180.000,B 0.000,C 180.000} C_DIS
LIN {X 111.021,Y 95.824,Z 70.500,A 180.000,B 0.000,C 180.000} C_DIS
LIN {X 110.945,Y 95.288,Z 70.500,A 180.000,B 0.000,C 180.000} C_DIS
LIN {X 110.914,Y 95.109,Z 70.500,A 180.000,B 0.000,C 180.000} C_DIS
LIN {X 110.807,Y 94.573,Z 70.500,A 180.000,B 0.000,C 180.000} C_DIS
LIN {X 110.766,Y 94.394,Z 70.500,A 180.000,B 0.000,C 180.000} C_DIS
LIN {X 110.720,Y 94.215,Z 70.500,A 180.000,B 0.000,C 180.000} C_DIS
LIN {X 110.628,Y 93.857,Z 70.500,A 180.000,B 0.000,C 180.000} C_DIS
LIN {X 110.579,Y 93.679,Z 70.500,A 180.000,B 0.000,C 180.000} C_DIS
LIN {X 110.523,Y 93.500,Z 70.500,A 180.000,B 0.000,C 180.000} C_DIS
LIN {X 110.502,Y 93.434,Z 70.500,A 180.000,B 0.000,C 180.000} C_DIS
; Link Move Starts
LIN {X 110.407,Y 93.135,Z 70.499,A 180.000,B 0.000,C 180.000} C_DIS
LIN {X 110.305,Y 92.844,Z 70.496,A 180.000,B 0.000,C 180.000} C_DIS
LIN {X 110.196,Y 92.551,Z 70.492,A 180.000,B 0.000,C 180.000} C_DIS
LIN {X 110.142,Y 92.406,Z 70.489,A 180.000,B 0.000,C 180.000} C_DIS
LIN {X 110.087,Y 92.262,Z 70.486,A 180.000,B 0.000,C 180.000} C_DIS
LIN {X 110.025,Y 92.119,Z 70.483,A 180.000,B 0.000,C 180.000} C_DIS
LIN {X 109.963,Y 91.975,Z 70.479,A 180.000,B 0.000,C 180.000} C_DIS
LIN {X 109.901,Y 91.832,Z 70.475,A 180.000,B 0.000,C 180.000} C_DIS
LIN {X 109.839,Y 91.688,Z 70.470,A 180.000,B 0.000,C 180.000} C_DIS
LIN {X 109.775,Y 91.547,Z 70.466,A 180.000,B 0.000,C 180.000} C_DIS
LIN {X 109.706,Y 91.409,Z 70.461,A 180.000,B 0.000,C 180.000} C_DIS
LIN {X 109.672,Y 91.339,Z 70.458,A 180.000,B 0.000,C 180.000} C_DIS
LIN {X 109.637,Y 91.269,Z 70.456,A 180.000,B 0.000,C 180.000} C_DIS
LIN {X 109.602,Y 91.199,Z 70.453,A 180.000,B 0.000,C 180.000} C_DIS
LIN {X 109.567,Y 91.128,Z 70.450,A 180.000,B 0.000,C 180.000} C_DIS
LIN {X 109.533,Y 91.059,Z 70.448,A 180.000,B 0.000,C 180.000} C_DIS
LIN {X 109.498,Y 90.990,Z 70.445,A 180.000,B 0.000,C 180.000} C_DIS
LIN {X 109.463,Y 90.921,Z 70.442,A 180.000,B 0.000,C 180.000} C_DIS
LIN {X 109.427,Y 90.853,Z 70.440,A 180.000,B 0.000,C 180.000} C_DIS
LIN {X 109.389,Y 90.785,Z 70.437,A 180.000,B 0.000,C 180.000} C_DIS
LIN {X 109.350,Y 90.717,Z 70.434,A 180.000,B 0.000,C 180.000} C_DIS
LIN {X 109.311,Y 90.649,Z 70.431,A 180.000,B 0.000,C 180.000} C_DIS
LIN {X 109.273,Y 90.580,Z 70.429,A 180.000,B 0.000,C 180.000} C_DIS
LIN {X 109.234,Y 90.513,Z 70.426,A 180.000,B 0.000,C 180.000} C_DIS
LIN {X 109.196,Y 90.445,Z 70.423,A 180.000,B 0.000,C 180.000} C_DIS
LIN {X 109.157,Y 90.377,Z 70.421,A 180.000,B 0.000,C 180.000} C_DIS
LIN {X 109.119,Y 90.309,Z 70.418,A 180.000,B 0.000,C 180.000} C_DIS
LIN {X 109.080,Y 90.242,Z 70.415,A 180.000,B 0.000,C 180.000} C_DIS
LIN {X 109.039,Y 90.176,Z 70.412,A 180.000,B 0.000,C 180.000} C_DIS
LIN {X 108.997,Y 90.110,Z 70.410,A 180.000,B 0.000,C 180.000} C_DIS
LIN {X 108.954,Y 90.045,Z 70.407,A 180.000,B 0.000,C 180.000} C_DIS
LIN {X 108.869,Y 89.913,Z 70.401,A 180.000,B 0.000,C 180.000} C_DIS
LIN {X 108.742,Y 89.716,Z 70.393,A 180.000,B 0.000,C 180.000} C_DIS
LIN {X 108.700,Y 89.651,Z 70.391,A 180.000,B 0.000,C 180.000} C_DIS
LIN {X 108.657,Y 89.587,Z 70.388,A 180.000,B 0.000,C 180.000} C_DIS
LIN {X 108.612,Y 89.523,Z 70.385,A 180.000,B 0.000,C 180.000} C_DIS
LIN {X 108.566,Y 89.460,Z 70.382,A 180.000,B 0.000,C 180.000} C_DIS
LIN {X 108.244,Y 89.017,Z 70.363,A 180.000,B 0.000,C 180.000} C_DIS
LIN {X 108.198,Y 88.955,Z 70.360,A 180.000,B 0.000,C 180.000} C_DIS
LIN {X 108.149,Y 88.894,Z 70.358,A 180.000,B 0.000,C 180.000} C_DIS
LIN {X 108.001,Y 88.712,Z 70.350,A 180.000,B 0.000,C 180.000} C_DIS
LIN {X 107.901,Y 88.591,Z 70.344,A 180.000,B 0.000,C 180.000} C_DIS
LIN {X 107.852,Y 88.530,Z 70.341,A 180.000,B 0.000,C 180.000} C_DIS
LIN {X 107.803,Y 88.470,Z 70.339,A 180.000,B 0.000,C 180.000} C_DIS
LIN {X 107.753,Y 88.409,Z 70.336,A 180.000,B 0.000,C 180.000} C_DIS
LIN {X 107.702,Y 88.350,Z 70.333,A 180.000,B 0.000,C 180.000} C_DIS
LIN {X 107.650,Y 88.293,Z 70.331,A 180.000,B 0.000,C 180.000} C_DIS
LIN {X 107.597,Y 88.235,Z 70.328,A 180.000,B 0.000,C 180.000} C_DIS
LIN {X 107.544,Y 88.177,Z 70.325,A 180.000,B 0.000,C 180.000} C_DIS
LIN {X 107.491,Y 88.119,Z 70.322,A 180.000,B 0.000,C 180.000} C_DIS
LIN {X 107.438,Y 88.061,Z 70.320,A 180.000,B 0.000,C 180.000} C_DIS
LIN {X 107.385,Y 88.004,Z 70.317,A 180.000,B 0.000,C 180.000} C_DIS
LIN {X 107.332,Y 87.946,Z 70.314,A 180.000,B 0.000,C 180.000} C_DIS
LIN {X 107.280,Y 87.888,Z 70.311,A 180.000,B 0.000,C 180.000} C_DIS
LIN {X 107.227,Y 87.830,Z 70.309,A 180.000,B 0.000,C 180.000} C_DIS
LIN {X 107.173,Y 87.774,Z 70.306,A 180.000,B 0.000,C 180.000} C_DIS
LIN {X 107.117,Y 87.719,Z 70.303,A 180.000,B 0.000,C 180.000} C_DIS
LIN {X 107.061,Y 87.665,Z 70.300,A 180.000,B 0.000,C 180.000} C_DIS
LIN {X 107.005,Y 87.610,Z 70.298,A 180.000,B 0.000,C 180.000} C_DIS
LIN {X 106.949,Y 87.555,Z 70.295,A 180.000,B 0.000,C 180.000} C_DIS
LIN {X 106.893,Y 87.500,Z 70.292,A 180.000,B 0.000,C 180.000} C_DIS
LIN {X 106.837,Y 87.446,Z 70.290,A 180.000,B 0.000,C 180.000} C_DIS
LIN {X 106.781,Y 87.391,Z 70.287,A 180.000,B 0.000,C 180.000} C_DIS
LIN {X 106.668,Y 87.282,Z 70.282,A 180.000,B 0.000,C 180.000} C_DIS
LIN {X 106.551,Y 87.178,Z 70.277,A 180.000,B 0.000,C 180.000} C_DIS
LIN {X 106.433,Y 87.076,Z 70.273,A 180.000,B 0.000,C 180.000} C_DIS
LIN {X 106.314,Y 86.973,Z 70.269,A 180.000,B 0.000,C 180.000} C_DIS
LIN {X 106.196,Y 86.870,Z 70.265,A 180.000,B 0.000,C 180.000} C_DIS
LIN {X 106.077,Y 86.769,Z 70.261,A 180.000,B 0.000,C 180.000} C_DIS
LIN {X 105.953,Y 86.672,Z 70.258,A 180.000,B 0.000,C 180.000} C_DIS
LIN {X 105.829,Y 86.576,Z 70.255,A 180.000,B 0.000,C 180.000} C_DIS
LIN {X 105.580,Y 86.386,Z 70.251,A 180.000,B 0.000,C 180.000} C_DIS
LIN {X 105.325,Y 86.204,Z 70.248,A 180.000,B 0.000,C 180.000} C_DIS
LIN {X 105.064,Y 86.029,Z 70.247,A 180.000,B 0.000,C 180.000} C_DIS
LIN {X 105.039,Y 86.015,Z 70.247,A 180.000,B 0.000,C 180.000} C_DIS
; Cutting Move Starts
LIN {X 104.941,Y 85.950,Z 70.247,A 180.000,B 0.000,C 180.000} C_DIS
LIN {X 104.762,Y 85.834,Z 70.247,A 180.000,B 0.000,C 180.000} C_DIS
LIN {X 104.727,Y 85.813,Z 70.247,A 180.000,B 0.000,C 180.000} C_DIS
LIN {X 104.226,Y 85.517,Z 70.247,A 180.000,B 0.000,C 180.000} C_DIS
LIN {X 104.116,Y 85.455,Z 70.247,A 180.000,B 0.000,C 180.000} C_DIS
LIN {X 104.047,Y 85.419,Z 70.247,A 180.000,B 0.000,C 180.000} C_DIS
LIN {X 103.690,Y 85.235,Z 70.247,A 180.000,B 0.000,C 180.000} C_DIS
LIN {X 103.511,Y 85.143,Z 70.247,A 180.000,B 0.000,C 180.000} C_DIS
LIN {X 103.417,Y 85.098,Z 70.247,A 180.000,B 0.000,C 180.000} C_DIS
LIN {X 103.332,Y 85.059,Z 70.247,A 180.000,B 0.000,C 180.000} C_DIS
LIN {X 102.975,Y 84.899,Z 70.247,A 180.000,B 0.000,C 180.000} C_DIS
LIN {X 102.796,Y 84.819,Z 70.247,A 180.000,B 0.000,C 180.000} C_DIS
LIN {X 102.617,Y 84.748,Z 70.247,A 180.000,B 0.000,C 180.000} C_DIS
LIN {X 102.128,Y 84.561,Z 70.247,A 180.000,B 0.000,C 180.000} C_DIS
LIN {X 102.081,Y 84.544,Z 70.247,A 180.000,B 0.000,C 180.000} C_DIS
LIN {X 101.902,Y 84.484,Z 70.247,A 180.000,B 0.000,C 180.000} C_DIS
LIN {X 101.366,Y 84.314,Z 70.247,A 180.000,B 0.000,C 180.000} C_DIS
LIN {X 101.187,Y 84.263,Z 70.247,A 180.000,B 0.000,C 180.000} C_DIS
LIN {X 100.651,Y 84.125,Z 70.247,A 180.000,B 0.000,C 180.000} C_DIS
LIN {X 100.472,Y 84.084,Z 70.247,A 180.000,B 0.000,C 180.000} C_DIS
LIN {X 99.936,Y 83.978,Z 70.247,A 180.000,B 0.000,C 180.000} C_DIS
LIN {X 99.757,Y 83.944,Z 70.247,A 180.000,B 0.000,C 180.000} C_DIS
LIN {X 99.578,Y 83.919,Z 70.247,A 180.000,B 0.000,C 180.000} C_DIS
LIN {X 99.221,Y 83.868,Z 70.247,A 180.000,B 0.000,C 180.000} C_DIS
LIN {X 99.060,Y 83.846,Z 70.247,A 180.000,B 0.000,C 180.000} C_DIS
LIN {X 99.042,Y 83.844,Z 70.247,A 180.000,B 0.000,C 180.000} C_DIS
LIN {X 98.863,Y 83.828,Z 70.247,A 180.000,B 0.000,C 180.000} C_DIS
LIN {X 98.505,Y 83.798,Z 70.247,A 180.000,B 0.000,C 180.000} C_DIS
LIN {X 98.327,Y 83.783,Z 70.247,A 180.000,B 0.000,C 180.000} C_DIS
LIN {X 98.148,Y 83.775,Z 70.247,A 180.000,B 0.000,C 180.000} C_DIS
LIN {X 97.612,Y 83.760,Z 70.247,A 180.000,B 0.000,C 180.000} C_DIS
LIN {X 97.433,Y 83.758,Z 70.247,A 180.000,B 0.000,C 180.000} C_DIS
LIN {X 96.897,Y 83.773,Z 70.247,A 180.000,B 0.000,C 180.000} C_DIS
LIN {X 96.718,Y 83.780,Z 70.247,A 180.000,B 0.000,C 180.000} C_DIS
LIN {X 96.539,Y 83.794,Z 70.247,A 180.000,B 0.000,C 180.000} C_DIS
LIN {X 96.181,Y 83.824,Z 70.247,A 180.000,B 0.000,C 180.000} C_DIS
LIN {X 96.003,Y 83.840,Z 70.247,A 180.000,B 0.000,C 180.000} C_DIS
LIN {X 95.940,Y 83.846,Z 70.247,A 180.000,B 0.000,C 180.000} C_DIS
LIN {X 95.824,Y 83.862,Z 70.247,A 180.000,B 0.000,C 180.000} C_DIS
LIN {X 95.288,Y 83.938,Z 70.247,A 180.000,B 0.000,C 180.000} C_DIS
LIN {X 95.109,Y 83.969,Z 70.247,A 180.000,B 0.000,C 180.000} C_DIS
LIN {X 94.573,Y 84.075,Z 70.247,A 180.000,B 0.000,C 180.000} C_DIS
LIN {X 94.394,Y 84.114,Z 70.247,A 180.000,B 0.000,C 180.000} C_DIS
LIN {X 94.215,Y 84.159,Z 70.247,A 180.000,B 0.000,C 180.000} C_DIS
LIN {X 93.857,Y 84.252,Z 70.247,A 180.000,B 0.000,C 180.000} C_DIS
LIN {X 93.679,Y 84.300,Z 70.247,A 180.000,B 0.000,C 180.000} C_DIS
LIN {X 93.500,Y 84.356,Z 70.247,A 180.000,B 0.000,C 180.000} C_DIS
LIN {X 93.142,Y 84.470,Z 70.247,A 180.000,B 0.000,C 180.000} C_DIS
LIN {X 92.964,Y 84.528,Z 70.247,A 180.000,B 0.000,C 180.000} C_DIS
LIN {X 92.872,Y 84.561,Z 70.247,A 180.000,B 0.000,C 180.000} C_DIS
LIN {X 92.404,Y 84.740,Z 70.247,A 180.000,B 0.000,C 180.000} C_DIS
LIN {X 92.249,Y 84.800,Z 70.247,A 180.000,B 0.000,C 180.000} C_DIS
LIN {X 92.070,Y 84.879,Z 70.247,A 180.000,B 0.000,C 180.000} C_DIS
LIN {X 91.712,Y 85.039,Z 70.247,A 180.000,B 0.000,C 180.000} C_DIS
LIN {X 91.583,Y 85.098,Z 70.247,A 180.000,B 0.000,C 180.000} C_DIS
LIN {X 91.533,Y 85.121,Z 70.247,A 180.000,B 0.000,C 180.000} C_DIS
LIN {X 91.355,Y 85.212,Z 70.247,A 180.000,B 0.000,C 180.000} C_DIS
LIN {X 90.997,Y 85.396,Z 70.247,A 180.000,B 0.000,C 180.000} C_DIS
LIN {X 90.884,Y 85.455,Z 70.247,A 180.000,B 0.000,C 180.000} C_DIS
LIN {X 90.818,Y 85.491,Z 70.247,A 180.000,B 0.000,C 180.000} C_DIS
LIN {X 90.640,Y 85.597,Z 70.247,A 180.000,B 0.000,C 180.000} C_DIS
LIN {X 90.273,Y 85.813,Z 70.247,A 180.000,B 0.000,C 180.000} C_DIS
LIN {X 90.103,Y 85.920,Z 70.247,A 180.000,B 0.000,C 180.000} C_DIS
LIN {X 89.728,Y 86.170,Z 70.247,A 180.000,B 0.000,C 180.000} C_DIS
LIN {X 89.567,Y 86.279,Z 70.247,A 180.000,B 0.000,C 180.000} C_DIS
LIN {X 89.470,Y 86.349,Z 70.247,A 180.000,B 0.000,C 180.000} C_DIS
LIN {X 88.995,Y 86.707,Z 70.247,A 180.000,B 0.000,C 180.000} C_DIS
LIN {X 88.852,Y 86.822,Z 70.247,A 180.000,B 0.000,C 180.000} C_DIS
LIN {X 88.494,Y 87.124,Z 70.247,A 180.000,B 0.000,C 180.000} C_DIS
LIN {X 88.354,Y 87.243,Z 70.247,A 180.000,B 0.000,C 180.000} C_DIS
LIN {X 88.316,Y 87.278,Z 70.247,A 180.000,B 0.000,C 180.000} C_DIS
LIN {X 88.163,Y 87.422,Z 70.247,A 180.000,B 0.000,C 180.000} C_DIS
LIN {X 87.958,Y 87.615,Z 70.247,A 180.000,B 0.000,C 180.000} C_DIS
LIN {X 87.786,Y 87.779,Z 70.247,A 180.000,B 0.000,C 180.000} C_DIS
LIN {X 87.779,Y 87.786,Z 70.247,A 180.000,B 0.000,C 180.000} C_DIS
LIN {X 87.616,Y 87.958,Z 70.247,A 180.000,B 0.000,C 180.000} C_DIS
LIN {X 87.422,Y 88.163,Z 70.247,A 180.000,B 0.000,C 180.000} C_DIS
LIN {X 87.278,Y 88.316,Z 70.247,A 180.000,B 0.000,C 180.000} C_DIS
LIN {X 87.243,Y 88.354,Z 70.247,A 180.000,B 0.000,C 180.000} C_DIS
LIN {X 87.124,Y 88.494,Z 70.247,A 180.000,B 0.000,C 180.000} C_DIS
LIN {X 86.822,Y 88.852,Z 70.247,A 180.000,B 0.000,C 180.000} C_DIS
LIN {X 86.707,Y 88.996,Z 70.247,A 180.000,B 0.000,C 180.000} C_DIS
LIN {X 86.349,Y 89.471,Z 70.247,A 180.000,B 0.000,C 180.000} C_DIS
LIN {X 86.279,Y 89.567,Z 70.247,A 180.000,B 0.000,C 180.000} C_DIS
LIN {X 86.170,Y 89.728,Z 70.247,A 180.000,B 0.000,C 180.000} C_DIS
LIN {X 85.920,Y 90.103,Z 70.247,A 180.000,B 0.000,C 180.000} C_DIS
LIN {X 85.813,Y 90.273,Z 70.247,A 180.000,B 0.000,C 180.000} C_DIS
LIN {X 85.597,Y 90.640,Z 70.247,A 180.000,B 0.000,C 180.000} C_DIS
LIN {X 85.492,Y 90.818,Z 70.247,A 180.000,B 0.000,C 180.000} C_DIS
LIN {X 85.455,Y 90.885,Z 70.247,A 180.000,B 0.000,C 180.000} C_DIS
LIN {X 85.396,Y 90.997,Z 70.247,A 180.000,B 0.000,C 180.000} C_DIS
LIN {X 85.212,Y 91.355,Z 70.247,A 180.000,B 0.000,C 180.000} C_DIS
LIN {X 85.120,Y 91.533,Z 70.247,A 180.000,B 0.000,C 180.000} C_DIS
LIN {X 85.098,Y 91.581,Z 70.247,A 180.000,B 0.000,C 180.000} C_DIS
LIN {X 85.039,Y 91.712,Z 70.247,A 180.000,B 0.000,C 180.000} C_DIS
LIN {X 84.879,Y 92.070,Z 70.247,A 180.000,B 0.000,C 180.000} C_DIS
LIN {X 84.801,Y 92.249,Z 70.247,A 180.000,B 0.000,C 180.000} C_DIS
LIN {X 84.740,Y 92.405,Z 70.247,A 180.000,B 0.000,C 180.000} C_DIS
LIN {X 84.561,Y 92.873,Z 70.247,A 180.000,B 0.000,C 180.000} C_DIS
LIN {X 84.528,Y 92.964,Z 70.247,A 180.000,B 0.000,C 180.000} C_DIS
LIN {X 84.470,Y 93.142,Z 70.247,A 180.000,B 0.000,C 180.000} C_DIS
LIN {X 84.356,Y 93.500,Z 70.247,A 180.000,B 0.000,C 180.000} C_DIS
LIN {X 84.300,Y 93.679,Z 70.247,A 180.000,B 0.000,C 180.000} C_DIS
LIN {X 84.252,Y 93.857,Z 70.247,A 180.000,B 0.000,C 180.000} C_DIS
LIN {X 84.160,Y 94.215,Z 70.247,A 180.000,B 0.000,C 180.000} C_DIS
LIN {X 84.114,Y 94.394,Z 70.247,A 180.000,B 0.000,C 180.000} C_DIS
LIN {X 84.075,Y 94.573,Z 70.247,A 180.000,B 0.000,C 180.000} C_DIS
LIN {X 83.968,Y 95.109,Z 70.247,A 180.000,B 0.000,C 180.000} C_DIS
LIN {X 83.938,Y 95.288,Z 70.247,A 180.000,B 0.000,C 180.000} C_DIS
LIN {X 83.863,Y 95.824,Z 70.247,A 180.000,B 0.000,C 180.000} C_DIS
LIN {X 83.846,Y 95.945,Z 70.247,A 180.000,B 0.000,C 180.000} C_DIS
LIN {X 83.840,Y 96.003,Z 70.247,A 180.000,B 0.000,C 180.000} C_DIS
LIN {X 83.824,Y 96.181,Z 70.247,A 180.000,B 0.000,C 180.000} C_DIS
LIN {X 83.794,Y 96.539,Z 70.247,A 180.000,B 0.000,C 180.000} C_DIS
LIN {X 83.780,Y 96.718,Z 70.247,A 180.000,B 0.000,C 180.000} C_DIS
LIN {X 83.773,Y 96.897,Z 70.247,A 180.000,B 0.000,C 180.000} C_DIS
LIN {X 83.763,Y 97.254,Z 70.247,A 180.000,B 0.000,C 180.000} C_DIS
LIN {X 83.759,Y 97.433,Z 70.247,A 180.000,B 0.000,C 180.000} C_DIS
LIN {X 83.760,Y 97.612,Z 70.247,A 180.000,B 0.000,C 180.000} C_DIS
LIN {X 83.775,Y 98.148,Z 70.247,A 180.000,B 0.000,C 180.000} C_DIS
LIN {X 83.783,Y 98.327,Z 70.247,A 180.000,B 0.000,C 180.000} C_DIS
LIN {X 83.798,Y 98.505,Z 70.247,A 180.000,B 0.000,C 180.000} C_DIS
LIN {X 83.828,Y 98.863,Z 70.247,A 180.000,B 0.000,C 180.000} C_DIS
LIN {X 83.845,Y 99.042,Z 70.247,A 180.000,B 0.000,C 180.000} C_DIS
LIN {X 83.846,Y 99.055,Z 70.247,A 180.000,B 0.000,C 180.000} C_DIS
LIN {X 83.869,Y 99.221,Z 70.247,A 180.000,B 0.000,C 180.000} C_DIS
LIN {X 83.919,Y 99.578,Z 70.247,A 180.000,B 0.000,C 180.000} C_DIS
LIN {X 83.945,Y 99.757,Z 70.247,A 180.000,B 0.000,C 180.000} C_DIS
LIN {X 83.977,Y 99.936,Z 70.247,A 180.000,B 0.000,C 180.000} C_DIS
LIN {X 84.084,Y 100.472,Z 70.247,A 180.000,B 0.000,C 180.000} C_DIS
LIN {X 84.125,Y 100.651,Z 70.247,A 180.000,B 0.000,C 180.000} C_DIS
LIN {X 84.264,Y 101.187,Z 70.247,A 180.000,B 0.000,C 180.000} C_DIS
LIN {X 84.313,Y 101.366,Z 70.247,A 180.000,B 0.000,C 180.000} C_DIS
LIN {X 84.370,Y 101.545,Z 70.247,A 180.000,B 0.000,C 180.000} C_DIS
LIN {X 84.484,Y 101.902,Z 70.247,A 180.000,B 0.000,C 180.000} C_DIS
LIN {X 84.544,Y 102.081,Z 70.247,A 180.000,B 0.000,C 180.000} C_DIS
LIN {X 84.561,Y 102.127,Z 70.247,A 180.000,B 0.000,C 180.000} C_DIS
LIN {X 84.749,Y 102.617,Z 70.247,A 180.000,B 0.000,C 180.000} C_DIS
LIN {X 84.819,Y 102.796,Z 70.247,A 180.000,B 0.000,C 180.000} C_DIS
LIN {X 84.899,Y 102.975,Z 70.247,A 180.000,B 0.000,C 180.000} C_DIS
LIN {X 85.059,Y 103.332,Z 70.247,A 180.000,B 0.000,C 180.000} C_DIS
LIN {X 85.098,Y 103.419,Z 70.247,A 180.000,B 0.000,C 180.000} C_DIS
LIN {X 85.142,Y 103.511,Z 70.247,A 180.000,B 0.000,C 180.000} C_DIS
LIN {X 85.235,Y 103.690,Z 70.247,A 180.000,B 0.000,C 180.000} C_DIS
LIN {X 85.419,Y 104.047,Z 70.247,A 180.000,B 0.000,C 180.000} C_DIS
LIN {X 85.455,Y 104.115,Z 70.247,A 180.000,B 0.000,C 180.000} C_DIS
LIN {X 85.517,Y 104.226,Z 70.247,A 180.000,B 0.000,C 180.000} C_DIS
LIN {X 85.813,Y 104.727,Z 70.247,A 180.000,B 0.000,C 180.000} C_DIS
LIN {X 85.834,Y 104.762,Z 70.247,A 180.000,B 0.000,C 180.000} C_DIS
LIN {X 85.949,Y 104.941,Z 70.247,A 180.000,B 0.000,C 180.000} C_DIS
LIN {X 86.188,Y 105.299,Z 70.247,A 180.000,B 0.000,C 180.000} C_DIS
LIN {X 86.311,Y 105.477,Z 70.247,A 180.000,B 0.000,C 180.000} C_DIS
LIN {X 86.349,Y 105.529,Z 70.247,A 180.000,B 0.000,C 180.000} C_DIS
LIN {X 86.714,Y 106.014,Z 70.247,A 180.000,B 0.000,C 180.000} C_DIS
LIN {X 86.859,Y 106.193,Z 70.247,A 180.000,B 0.000,C 180.000} C_DIS
LIN {X 87.161,Y 106.550,Z 70.247,A 180.000,B 0.000,C 180.000} C_DIS
LIN {X 87.243,Y 106.646,Z 70.247,A 180.000,B 0.000,C 180.000} C_DIS
LIN {X 87.320,Y 106.729,Z 70.247,A 180.000,B 0.000,C 180.000} C_DIS
LIN {X 87.658,Y 107.086,Z 70.247,A 180.000,B 0.000,C 180.000} C_DIS
LIN {X 87.779,Y 107.214,Z 70.247,A 180.000,B 0.000,C 180.000} C_DIS
LIN {X 87.832,Y 107.265,Z 70.247,A 180.000,B 0.000,C 180.000} C_DIS
LIN {X 87.958,Y 107.385,Z 70.247,A 180.000,B 0.000,C 180.000} C_DIS
LIN {X 88.210,Y 107.623,Z 70.247,A 180.000,B 0.000,C 180.000} C_DIS
LIN {X 88.316,Y 107.722,Z 70.247,A 180.000,B 0.000,C 180.000} C_DIS
LIN {X 88.406,Y 107.802,Z 70.247,A 180.000,B 0.000,C 180.000} C_DIS
LIN {X 88.852,Y 108.178,Z 70.247,A 180.000,B 0.000,C 180.000} C_DIS
LIN {X 89.031,Y 108.320,Z 70.247,A 180.000,B 0.000,C 180.000} C_DIS
LIN {X 89.388,Y 108.589,Z 70.247,A 180.000,B 0.000,C 180.000} C_DIS
LIN {X 89.530,Y 108.695,Z 70.247,A 180.000,B 0.000,C 180.000} C_DIS
LIN {X 89.567,Y 108.721,Z 70.247,A 180.000,B 0.000,C 180.000} C_DIS
LIN {X 89.746,Y 108.841,Z 70.247,A 180.000,B 0.000,C 180.000} C_DIS
LIN {X 90.103,Y 109.080,Z 70.247,A 180.000,B 0.000,C 180.000} C_DIS
LIN {X 90.282,Y 109.192,Z 70.247,A 180.000,B 0.000,C 180.000} C_DIS
LIN {X 90.652,Y 109.410,Z 70.247,A 180.000,B 0.000,C 180.000} C_DIS
LIN {X 90.818,Y 109.509,Z 70.247,A 180.000,B 0.000,C 180.000} C_DIS
LIN {X 90.969,Y 109.589,Z 70.247,A 180.000,B 0.000,C 180.000} C_DIS
LIN {X 91.355,Y 109.788,Z 70.247,A 180.000,B 0.000,C 180.000} C_DIS
LIN {X 91.533,Y 109.879,Z 70.247,A 180.000,B 0.000,C 180.000} C_DIS
LIN {X 91.681,Y 109.947,Z 70.247,A 180.000,B 0.000,C 180.000} C_DIS
LIN {X 92.080,Y 110.126,Z 70.247,A 180.000,B 0.000,C 180.000} C_DIS
LIN {X 92.249,Y 110.200,Z 70.247,A 180.000,B 0.000,C 180.000} C_DIS
LIN {X 92.427,Y 110.269,Z 70.247,A 180.000,B 0.000,C 180.000} C_DIS
LIN {X 92.785,Y 110.405,Z 70.247,A 180.000,B 0.000,C 180.000} C_DIS
LIN {X 92.964,Y 110.472,Z 70.247,A 180.000,B 0.000,C 180.000} C_DIS
LIN {X 92.997,Y 110.483,Z 70.247,A 180.000,B 0.000,C 180.000} C_DIS
LIN {X 93.142,Y 110.530,Z 70.247,A 180.000,B 0.000,C 180.000} C_DIS
LIN {X 93.557,Y 110.662,Z 70.247,A 180.000,B 0.000,C 180.000} C_DIS
LIN {X 93.679,Y 110.700,Z 70.247,A 180.000,B 0.000,C 180.000} C_DIS
LIN {X 93.857,Y 110.748,Z 70.247,A 180.000,B 0.000,C 180.000} C_DIS
LIN {X 94.215,Y 110.841,Z 70.247,A 180.000,B 0.000,C 180.000} C_DIS
LIN {X 94.394,Y 110.886,Z 70.247,A 180.000,B 0.000,C 180.000} C_DIS
LIN {X 94.573,Y 110.925,Z 70.247,A 180.000,B 0.000,C 180.000} C_DIS
LIN {X 95.049,Y 111.019,Z 70.247,A 180.000,B 0.000,C 180.000} C_DIS
LIN {X 95.109,Y 111.031,Z 70.247,A 180.000,B 0.000,C 180.000} C_DIS
LIN {X 95.288,Y 111.062,Z 70.247,A 180.000,B 0.000,C 180.000} C_DIS
LIN {X 95.824,Y 111.138,Z 70.247,A 180.000,B 0.000,C 180.000} C_DIS
LIN {X 96.003,Y 111.160,Z 70.247,A 180.000,B 0.000,C 180.000} C_DIS
LIN {X 96.181,Y 111.176,Z 70.247,A 180.000,B 0.000,C 180.000} C_DIS
LIN {X 96.539,Y 111.206,Z 70.247,A 180.000,B 0.000,C 180.000} C_DIS
LIN {X 96.718,Y 111.220,Z 70.247,A 180.000,B 0.000,C 180.000} C_DIS
LIN {X 96.897,Y 111.227,Z 70.247,A 180.000,B 0.000,C 180.000} C_DIS
LIN {X 97.433,Y 111.242,Z 70.247,A 180.000,B 0.000,C 180.000} C_DIS
LIN {X 97.612,Y 111.240,Z 70.247,A 180.000,B 0.000,C 180.000} C_DIS
LIN {X 98.148,Y 111.225,Z 70.247,A 180.000,B 0.000,C 180.000} C_DIS
LIN {X 98.327,Y 111.217,Z 70.247,A 180.000,B 0.000,C 180.000} C_DIS
LIN {X 98.505,Y 111.202,Z 70.247,A 180.000,B 0.000,C 180.000} C_DIS
LIN {X 98.863,Y 111.172,Z 70.247,A 180.000,B 0.000,C 180.000} C_DIS
LIN {X 99.042,Y 111.156,Z 70.247,A 180.000,B 0.000,C 180.000} C_DIS
LIN {X 99.221,Y 111.132,Z 70.247,A 180.000,B 0.000,C 180.000} C_DIS
LIN {X 99.578,Y 111.081,Z 70.247,A 180.000,B 0.000,C 180.000} C_DIS
LIN {X 99.757,Y 111.056,Z 70.247,A 180.000,B 0.000,C 180.000} C_DIS
LIN {X 99.936,Y 111.022,Z 70.247,A 180.000,B 0.000,C 180.000} C_DIS
LIN {X 100.472,Y 110.916,Z 70.247,A 180.000,B 0.000,C 180.000} C_DIS
LIN {X 100.651,Y 110.875,Z 70.247,A 180.000,B 0.000,C 180.000} C_DIS
LIN {X 101.187,Y 110.737,Z 70.247,A 180.000,B 0.000,C 180.000} C_DIS
LIN {X 101.366,Y 110.686,Z 70.247,A 180.000,B 0.000,C 180.000} C_DIS
LIN {X 101.902,Y 110.516,Z 70.247,A 180.000,B 0.000,C 180.000} C_DIS
LIN {X 102.003,Y 110.483,Z 70.247,A 180.000,B 0.000,C 180.000} C_DIS
LIN {X 102.081,Y 110.456,Z 70.247,A 180.000,B 0.000,C 180.000} C_DIS
LIN {X 102.260,Y 110.388,Z 70.247,A 180.000,B 0.000,C 180.000} C_DIS
LIN {X 102.617,Y 110.252,Z 70.247,A 180.000,B 0.000,C 180.000} C_DIS
LIN {X 102.796,Y 110.181,Z 70.247,A 180.000,B 0.000,C 180.000} C_DIS
LIN {X 102.920,Y 110.126,Z 70.247,A 180.000,B 0.000,C 180.000} C_DIS
LIN {X 103.332,Y 109.941,Z 70.247,A 180.000,B 0.000,C 180.000} C_DIS
LIN {X 103.511,Y 109.857,Z 70.247,A 180.000,B 0.000,C 180.000} C_DIS
LIN {X 103.685,Y 109.768,Z 70.247,A 180.000,B 0.000,C 180.000} C_DIS
LIN {X 104.047,Y 109.581,Z 70.247,A 180.000,B 0.000,C 180.000} C_DIS
LIN {X 104.226,Y 109.483,Z 70.247,A 180.000,B 0.000,C 180.000} C_DIS
LIN {X 104.651,Y 109.232,Z 70.247,A 180.000,B 0.000,C 180.000} C_DIS
LIN {X 104.762,Y 109.166,Z 70.247,A 180.000,B 0.000,C 180.000} C_DIS
LIN {X 104.938,Y 109.053,Z 70.247,A 180.000,B 0.000,C 180.000} C_DIS
LIN {X 105.299,Y 108.812,Z 70.247,A 180.000,B 0.000,C 180.000} C_DIS
LIN {X 105.470,Y 108.695,Z 70.247,A 180.000,B 0.000,C 180.000} C_DIS
LIN {X 105.477,Y 108.690,Z 70.247,A 180.000,B 0.000,C 180.000} C_DIS
LIN {X 105.656,Y 108.556,Z 70.247,A 180.000,B 0.000,C 180.000} C_DIS
LIN {X 105.946,Y 108.338,Z 70.247,A 180.000,B 0.000,C 180.000} C_DIS
LIN {X 106.014,Y 108.287,Z 70.247,A 180.000,B 0.000,C 180.000} C_DIS
LIN {X 106.170,Y 108.159,Z 70.247,A 180.000,B 0.000,C 180.000} C_DIS
LIN {X 106.594,Y 107.802,Z 70.247,A 180.000,B 0.000,C 180.000} C_DIS
LIN {X 106.729,Y 107.681,Z 70.247,A 180.000,B 0.000,C 180.000} C_DIS
LIN {X 107.086,Y 107.343,Z 70.247,A 180.000,B 0.000,C 180.000} C_DIS
LIN {X 107.168,Y 107.265,Z 70.247,A 180.000,B 0.000,C 180.000} C_DIS
LIN {X 107.265,Y 107.168,Z 70.247,A 180.000,B 0.000,C 180.000} C_DIS
LIN {X 107.680,Y 106.729,Z 70.247,A 180.000,B 0.000,C 180.000} C_DIS
LIN {X 107.802,Y 106.594,Z 70.247,A 180.000,B 0.000,C 180.000} C_DIS
LIN {X 108.159,Y 106.171,Z 70.247,A 180.000,B 0.000,C 180.000} C_DIS
LIN {X 108.286,Y 106.014,Z 70.247,A 180.000,B 0.000,C 180.000} C_DIS
LIN {X 108.555,Y 105.656,Z 70.247,A 180.000,B 0.000,C 180.000} C_DIS
LIN {X 108.689,Y 105.477,Z 70.247,A 180.000,B 0.000,C 180.000} C_DIS
LIN {X 108.695,Y 105.469,Z 70.247,A 180.000,B 0.000,C 180.000} C_DIS
LIN {X 108.812,Y 105.299,Z 70.247,A 180.000,B 0.000,C 180.000} C_DIS
LIN {X 109.053,Y 104.938,Z 70.247,A 180.000,B 0.000,C 180.000} C_DIS
LIN {X 109.166,Y 104.762,Z 70.247,A 180.000,B 0.000,C 180.000} C_DIS
LIN {X 109.232,Y 104.651,Z 70.247,A 180.000,B 0.000,C 180.000} C_DIS
LIN {X 109.483,Y 104.226,Z 70.247,A 180.000,B 0.000,C 180.000} C_DIS
LIN {X 109.581,Y 104.047,Z 70.247,A 180.000,B 0.000,C 180.000} C_DIS
LIN {X 109.768,Y 103.685,Z 70.247,A 180.000,B 0.000,C 180.000} C_DIS
LIN {X 109.858,Y 103.511,Z 70.247,A 180.000,B 0.000,C 180.000} C_DIS
LIN {X 109.941,Y 103.332,Z 70.247,A 180.000,B 0.000,C 180.000} C_DIS
LIN {X 110.126,Y 102.920,Z 70.247,A 180.000,B 0.000,C 180.000} C_DIS
LIN {X 110.181,Y 102.796,Z 70.247,A 180.000,B 0.000,C 180.000} C_DIS
LIN {X 110.251,Y 102.617,Z 70.247,A 180.000,B 0.000,C 180.000} C_DIS
LIN {X 110.388,Y 102.260,Z 70.247,A 180.000,B 0.000,C 180.000} C_DIS
LIN {X 110.456,Y 102.081,Z 70.247,A 180.000,B 0.000,C 180.000} C_DIS
LIN {X 110.483,Y 102.005,Z 70.247,A 180.000,B 0.000,C 180.000} C_DIS
LIN {X 110.516,Y 101.902,Z 70.247,A 180.000,B 0.000,C 180.000} C_DIS
LIN {X 110.662,Y 101.445,Z 70.247,A 180.000,B 0.000,C 180.000} C_DIS
LIN {X 110.687,Y 101.366,Z 70.247,A 180.000,B 0.000,C 180.000} C_DIS
LIN {X 110.736,Y 101.187,Z 70.247,A 180.000,B 0.000,C 180.000} C_DIS
LIN {X 110.875,Y 100.651,Z 70.247,A 180.000,B 0.000,C 180.000} C_DIS
LIN {X 110.916,Y 100.472,Z 70.247,A 180.000,B 0.000,C 180.000} C_DIS
LIN {X 111.023,Y 99.936,Z 70.247,A 180.000,B 0.000,C 180.000} C_DIS
LIN {X 111.055,Y 99.757,Z 70.247,A 180.000,B 0.000,C 180.000} C_DIS
LIN {X 111.081,Y 99.578,Z 70.247,A 180.000,B 0.000,C 180.000} C_DIS
LIN {X 111.131,Y 99.221,Z 70.247,A 180.000,B 0.000,C 180.000} C_DIS
LIN {X 111.155,Y 99.042,Z 70.247,A 180.000,B 0.000,C 180.000} C_DIS
LIN {X 111.172,Y 98.863,Z 70.247,A 180.000,B 0.000,C 180.000} C_DIS
LIN {X 111.202,Y 98.505,Z 70.247,A 180.000,B 0.000,C 180.000} C_DIS
LIN {X 111.217,Y 98.327,Z 70.247,A 180.000,B 0.000,C 180.000} C_DIS
LIN {X 111.225,Y 98.148,Z 70.247,A 180.000,B 0.000,C 180.000} C_DIS
LIN {X 111.240,Y 97.612,Z 70.247,A 180.000,B 0.000,C 180.000} C_DIS
LIN {X 111.241,Y 97.433,Z 70.247,A 180.000,B 0.000,C 180.000} C_DIS
LIN {X 111.237,Y 97.254,Z 70.247,A 180.000,B 0.000,C 180.000} C_DIS
LIN {X 111.227,Y 96.897,Z 70.247,A 180.000,B 0.000,C 180.000} C_DIS
LIN {X 111.220,Y 96.718,Z 70.247,A 180.000,B 0.000,C 180.000} C_DIS
LIN {X 111.206,Y 96.539,Z 70.247,A 180.000,B 0.000,C 180.000} C_DIS
LIN {X 111.176,Y 96.181,Z 70.247,A 180.000,B 0.000,C 180.000} C_DIS
LIN {X 111.160,Y 96.003,Z 70.247,A 180.000,B 0.000,C 180.000} C_DIS
LIN {X 111.137,Y 95.824,Z 70.247,A 180.000,B 0.000,C 180.000} C_DIS
LIN {X 111.062,Y 95.288,Z 70.247,A 180.000,B 0.000,C 180.000} C_DIS
LIN {X 111.032,Y 95.109,Z 70.247,A 180.000,B 0.000,C 180.000} C_DIS
LIN {X 110.925,Y 94.573,Z 70.247,A 180.000,B 0.000,C 180.000} C_DIS
LIN {X 110.886,Y 94.394,Z 70.247,A 180.000,B 0.000,C 180.000} C_DIS
LIN {X 110.840,Y 94.215,Z 70.247,A 180.000,B 0.000,C 180.000} C_DIS
LIN {X 110.748,Y 93.857,Z 70.247,A 180.000,B 0.000,C 180.000} C_DIS
LIN {X 110.700,Y 93.679,Z 70.247,A 180.000,B 0.000,C 180.000} C_DIS
LIN {X 110.662,Y 93.555,Z 70.247,A 180.000,B 0.000,C 180.000} C_DIS
LIN {X 110.530,Y 93.142,Z 70.247,A 180.000,B 0.000,C 180.000} C_DIS
LIN {X 110.483,Y 92.995,Z 70.247,A 180.000,B 0.000,C 180.000} C_DIS
LIN {X 110.472,Y 92.964,Z 70.247,A 180.000,B 0.000,C 180.000} C_DIS
LIN {X 110.405,Y 92.785,Z 70.247,A 180.000,B 0.000,C 180.000} C_DIS
LIN {X 110.268,Y 92.427,Z 70.247,A 180.000,B 0.000,C 180.000} C_DIS
LIN {X 110.199,Y 92.249,Z 70.247,A 180.000,B 0.000,C 180.000} C_DIS
LIN {X 110.126,Y 92.080,Z 70.247,A 180.000,B 0.000,C 180.000} C_DIS
LIN {X 109.947,Y 91.680,Z 70.247,A 180.000,B 0.000,C 180.000} C_DIS
LIN {X 109.880,Y 91.533,Z 70.247,A 180.000,B 0.000,C 180.000} C_DIS
LIN {X 109.788,Y 91.355,Z 70.247,A 180.000,B 0.000,C 180.000} C_DIS
LIN {X 109.589,Y 90.969,Z 70.247,A 180.000,B 0.000,C 180.000} C_DIS
LIN {X 109.508,Y 90.818,Z 70.247,A 180.000,B 0.000,C 180.000} C_DIS
LIN {X 109.410,Y 90.652,Z 70.247,A 180.000,B 0.000,C 180.000} C_DIS
LIN {X 109.192,Y 90.282,Z 70.247,A 180.000,B 0.000,C 180.000} C_DIS
LIN {X 109.080,Y 90.103,Z 70.247,A 180.000,B 0.000,C 180.000} C_DIS
LIN {X 108.841,Y 89.746,Z 70.247,A 180.000,B 0.000,C 180.000} C_DIS
LIN {X 108.721,Y 89.567,Z 70.247,A 180.000,B 0.000,C 180.000} C_DIS
LIN {X 108.695,Y 89.531,Z 70.247,A 180.000,B 0.000,C 180.000} C_DIS
LIN {X 108.589,Y 89.388,Z 70.247,A 180.000,B 0.000,C 180.000} C_DIS
LIN {X 108.320,Y 89.031,Z 70.247,A 180.000,B 0.000,C 180.000} C_DIS
LIN {X 108.178,Y 88.852,Z 70.247,A 180.000,B 0.000,C 180.000} C_DIS
LIN {X 107.802,Y 88.406,Z 70.247,A 180.000,B 0.000,C 180.000} C_DIS
LIN {X 107.722,Y 88.316,Z 70.247,A 180.000,B 0.000,C 180.000} C_DIS
LIN {X 107.623,Y 88.210,Z 70.247,A 180.000,B 0.000,C 180.000} C_DIS
LIN {X 107.265,Y 87.832,Z 70.247,A 180.000,B 0.000,C 180.000} C_DIS
LIN {X 107.214,Y 87.779,Z 70.247,A 180.000,B 0.000,C 180.000} C_DIS
LIN {X 107.086,Y 87.657,Z 70.247,A 180.000,B 0.000,C 180.000} C_DIS
LIN {X 106.729,Y 87.319,Z 70.247,A 180.000,B 0.000,C 180.000} C_DIS
LIN {X 106.646,Y 87.243,Z 70.247,A 180.000,B 0.000,C 180.000} C_DIS
LIN {X 106.550,Y 87.162,Z 70.247,A 180.000,B 0.000,C 180.000} C_DIS
LIN {X 106.193,Y 86.860,Z 70.247,A 180.000,B 0.000,C 180.000} C_DIS
LIN {X 106.014,Y 86.713,Z 70.247,A 180.000,B 0.000,C 180.000} C_DIS
LIN {X 106.005,Y 86.707,Z 70.247,A 180.000,B 0.000,C 180.000} C_DIS
LIN {X 105.530,Y 86.349,Z 70.247,A 180.000,B 0.000,C 180.000} C_DIS
LIN {X 105.477,Y 86.310,Z 70.247,A 180.000,B 0.000,C 180.000} C_DIS
LIN {X 105.299,Y 86.188,Z 70.247,A 180.000,B 0.000,C 180.000} C_DIS
LIN {X 105.039,Y 86.015,Z 70.247,A 180.000,B 0.000,C 180.000} C_DIS
; Link Move Starts
LIN {X 104.789,Y 85.847,Z 70.246,A 180.000,B 0.000,C 180.000} C_DIS
LIN {X 104.529,Y 85.692,Z 70.243,A 180.000,B 0.000,C 180.000} C_DIS
LIN {X 104.268,Y 85.535,Z 70.239,A 180.000,B 0.000,C 180.000} C_DIS
LIN {X 104.138,Y 85.459,Z 70.236,A 180.000,B 0.000,C 180.000} C_DIS
LIN {X 104.006,Y 85.388,Z 70.233,A 180.000,B 0.000,C 180.000} C_DIS
LIN {X 103.872,Y 85.317,Z 70.230,A 180.000,B 0.000,C 180.000} C_DIS
LIN {X 103.737,Y 85.246,Z 70.226,A 180.000,B 0.000,C 180.000} C_DIS
LIN {X 103.603,Y 85.174,Z 70.222,A 180.000,B 0.000,C 180.000} C_DIS
LIN {X 103.468,Y 85.104,Z 70.218,A 180.000,B 0.000,C 180.000} C_DIS
LIN {X 103.332,Y 85.040,Z 70.213,A 180.000,B 0.000,C 180.000} C_DIS
LIN {X 103.196,Y 84.976,Z 70.209,A 180.000,B 0.000,C 180.000} C_DIS
LIN {X 103.127,Y 84.944,Z 70.206,A 180.000,B 0.000,C 180.000} C_DIS
LIN {X 103.058,Y 84.912,Z 70.204,A 180.000,B 0.000,C 180.000} C_DIS
